LIN {X 0,Y 547.615,Z 386.436,A -85,B 0,C 180,E1 18147.997,E2 18147.997} C_VEL
LIN {X 0,Y 557.313,Z 399.518,A -85,B 0,C 180,E1 18145.988,E2 18145.988} C_VEL
LIN {X 0,Y 566.664,Z 412.794,A -85,B 0,C 180,E1 18144.201,E2 18144.201} C_VEL
LIN {X 0,Y 578.034,Z 429.679,A -85,B 0,C 180,E1 18142.193,E2 18142.193} C_VEL
LIN {X 0,Y 584.71,Z 440.377,A -85,B 0,C 180,E1 18141.078,E2 18141.078} C_VEL
LIN {X 0,Y 587.079,Z 454.76,A -85,B 0,C 180,E1 18140.491,E2 18140.491} C_VEL
LIN {X 0,Y 578.942,Z 687.19,A -85,B 0,C 180,E1 18137.176,E2 18137.176} C_VEL
LIN {X 0,Y 574.123,Z 831.147,A -85,B 0,C 180,E1 18135.139,E2 18135.139} C_VEL
LIN {X 0,Y 572.503,Z 855.718,A -85,B 0,C 180,E1 18134.679,E2 18134.679} C_VEL
LIN {X 0,Y 571.103,Z 863.307,A -85,B 0,C 180,E1 18134.585,E2 18134.585} C_VEL
LIN {X 0,Y 565.25,Z 881.378,A -85,B 0,C 180,E1 18134.516,E2 18134.516} C_VEL
LIN {X 0,Y 563.615,Z 888.829,A -85,B 0,C 180,E1 18134.375,E2 18134.375} C_VEL
LIN {X 0,Y 563.486,Z 889.888,A -85,B 0,C 180,E1 18134.344,E2 18134.344} C_VEL
LIN {X 0,Y 560.294,Z 914.057,A -85,B 0,C 180,E1 18133.468,E2 18133.468} C_VEL
LIN {X 0,Y 557.17,Z 934.515,A -85,B 0,C 180,E1 18132.575,E2 18132.575} C_VEL
LIN {X 0,Y 553.827,Z 954.3,A -85,B 0,C 180,E1 18131.566,E2 18131.566} C_VEL
LIN {X 0,Y 549.439,Z 977.967,A -85,B 0,C 180,E1 18130.152,E2 18130.152} C_VEL
LIN {X 0,Y 545.24,Z 998.451,A -85,B 0,C 180,E1 18128.707,E2 18128.707} C_VEL
LIN {X 0,Y 541.433,Z 1016.198,A -85,B 0,C 180,E1 18127.281,E2 18127.281} C_VEL
LIN {X 0,Y 536.891,Z 1036.776,A -85,B 0,C 180,E1 18125.394,E2 18125.394} C_VEL
LIN {X 0,Y 532.749,Z 1054.642,A -85,B 0,C 180,E1 18123.49,E2 18123.49} C_VEL
LIN {X 0,Y 529.257,Z 1069.696,A -85,B 0,C 180,E1 18121.682,E2 18121.682} C_VEL
LIN {X 0,Y 525.468,Z 1086.495,A -85,B 0,C 180,E1 18119.402,E2 18119.402} C_VEL
LIN {X 0,Y 522.072,Z 1101.673,A -85,B 0,C 180,E1 18116.995,E2 18116.995} C_VEL
LIN {X 0,Y 519.505,Z 1113.829,A -85,B 0,C 180,E1 18114.808,E2 18114.808} C_VEL
LIN {X 0,Y 517.039,Z 1126.95,A -85,B 0,C 180,E1 18112.13,E2 18112.13} C_VEL
LIN {X 0,Y 515.099,Z 1138.408,A -85,B 0,C 180,E1 18109.368,E2 18109.368} C_VEL
LIN {X 0,Y 513.904,Z 1147.043,A -85,B 0,C 180,E1 18106.969,E2 18106.969} C_VEL
LIN {X 0,Y 512.891,Z 1156.089,A -85,B 0,C 180,E1 18103.989,E2 18103.989} C_VEL
LIN {X 0,Y 512.347,Z 1162.485,A -85,B 0,C 180,E1 18101.368,E2 18101.368} C_VEL
LIN {X 0,Y 512.097,Z 1167.168,A -85,B 0,C 180,E1 18098.987,E2 18098.987} C_VEL
LIN {X 0,Y 511.954,Z 1171.379,A -85,B 0,C 180,E1 18096.167,E2 18096.167} C_VEL
LIN {X 0,Y 511.906,Z 1173.875,A -85,B 0,C 180,E1 18093.36,E2 18093.36} C_VEL
LIN {X 0,Y 511.909,Z 1174.869,A -85,B 0,C 180,E1 18091.007,E2 18091.007} C_VEL
LIN {X 0,Y 511.912,Z 1174.823,A -85,B 0,C 180,E1 18088.657,E2 18088.657} C_VEL
LIN {X 0,Y 511.915,Z 1173.467,A -85,B 0,C 180,E1 18085.856,E2 18085.856} C_VEL
LIN {X 0,Y 511.966,Z 1170.412,A -85,B 0,C 180,E1 18083.045,E2 18083.045} C_VEL
LIN {X 0,Y 512.119,Z 1166.721,A -85,B 0,C 180,E1 18080.674,E2 18080.674} C_VEL
LIN {X 0,Y 512.415,Z 1161.69,A -85,B 0,C 180,E1 18078.177,E2 18078.177} C_VEL
LIN {X 0,Y 513.117,Z 1153.749,A -85,B 0,C 180,E1 18075.095,E2 18075.095} C_VEL
LIN {X 0,Y 514.003,Z 1146.165,A -85,B 0,C 180,E1 18072.685,E2 18072.685} C_VEL
LIN {X 0,Y 515.264,Z 1137.342,A -85,B 0,C 180,E1 18070.267,E2 18070.267} C_VEL
LIN {X 0,Y 517.45,Z 1124.512,A -85,B 0,C 180,E1 18067.266,E2 18067.266} C_VEL
LIN {X 0,Y 519.656,Z 1113.054,A -85,B 0,C 180,E1 18064.957,E2 18064.957} C_VEL
LIN {X 0,Y 522.419,Z 1100.156,A -85,B 0,C 180,E1 18062.655,E2 18062.655} C_VEL
LIN {X 0,Y 526.146,Z 1083.341,A -85,B 0,C 180,E1 18060.065,E2 18060.065} C_VEL
LIN {X 0,Y 529.53,Z 1068.546,A -85,B 0,C 180,E1 18058.082,E2 18058.082} C_VEL
LIN {X 0,Y 533.173,Z 1052.881,A -85,B 0,C 180,E1 18056.218,E2 18056.218} C_VEL
LIN {X 0,Y 537.976,Z 1031.771,A -85,B 0,C 180,E1 18054.034,E2 18054.034} C_VEL
LIN {X 0,Y 541.945,Z 1013.857,A -85,B 0,C 180,E1 18052.428,E2 18052.428} C_VEL
LIN {X 0,Y 546.122,Z 994.411,A -85,B 0,C 180,E1 18050.895,E2 18050.895} C_VEL
LIN {X 0,Y 550.757,Z 971.131,A -85,B 0,C 180,E1 18049.327,E2 18049.327} C_VEL
LIN {X 0,Y 554.306,Z 951.689,A -85,B 0,C 180,E1 18048.202,E2 18048.202} C_VEL
LIN {X 0,Y 557.851,Z 930.54,A -85,B 0,C 180,E1 18047.146,E2 18047.146} C_VEL
LIN {X 0,Y 561.578,Z 905.044,A -85,B 0,C 180,E1 18046.093,E2 18046.093} C_VEL
LIN {X 0,Y 564.218,Z 883.465,A -85,B 0,C 180,E1 18045.369,E2 18045.369} C_VEL
LIN {X 0,Y 566.449,Z 861.689,A -85,B 0,C 180,E1 18044.778,E2 18044.778} C_VEL
LIN {X 0,Y 568.589,Z 834.181,A -85,B 0,C 180,E1 18044.222,E2 18044.222} C_VEL
LIN {X 0,Y 570.674,Z 778.593,A -85,B 0,C 180,E1 18043.415,E2 18043.415} C_VEL
LIN {X 0,Y 578.51,Z 553.659,A -85,B 0,C 180,E1 18040.214,E2 18040.214} C_VEL
LIN {X 0,Y 582.134,Z 455.512,A -85,B 0,C 180,E1 18038.781,E2 18038.781} C_VEL
LIN {X 0,Y 580.157,Z 444.764,A -85,B 0,C 180,E1 18038.302,E2 18038.302} C_VEL
LIN {X 0,Y 568.568,Z 426.659,A -85,B 0,C 180,E1 18036.283,E2 18036.283} C_VEL
LIN {X 0,Y 557.682,Z 410.932,A -85,B 0,C 180,E1 18034.232,E2 18034.232} C_VEL
LIN {X 0,Y 548.268,Z 397.906,A -85,B 0,C 180,E1 18032.3,E2 18032.3} C_VEL
LIN {X 0,Y 538.549,Z 384.76,A -85,B 0,C 180,E1 18030.086,E2 18030.086} C_VEL
LIN {X 0,Y 533.593,Z 375.407,A -85,B 0,C 180,E1 18027.814,E2 18027.814} C_VEL
LIN {X 0,Y 530.924,Z 370.532,A -85,B 0,C 180,E1 18026.509,E2 18026.509} C_VEL
LIN {X 0,Y 528.411,Z 365.874,A -85,B 0,C 180,E1 18025.199,E2 18025.199} C_VEL
LIN {X 0,Y 525.594,Z 360.858,A -85,B 0,C 180,E1 18023.666,E2 18023.666} C_VEL
LIN {X 0,Y 522.985,Z 356.145,A -85,B 0,C 180,E1 18022.126,E2 18022.126} C_VEL
LIN {X 0,Y 520.688,Z 352.401,A -85,B 0,C 180,E1 18020.743,E2 18020.743} C_VEL
LIN {X 0,Y 519.792,Z 350.773,A -85,B 0,C 180,E1 18020.141,E2 18020.141} C_VEL
LIN {X 0,Y 517.475,Z 347.05,A -85,B 0,C 180,E1 18018.592,E2 18018.592} C_VEL
LIN {X 0,Y 516.625,Z 345.409,A -85,B 0,C 180,E1 18017.923,E2 18017.923} C_VEL
LIN {X 0,Y 514.179,Z 341.868,A -85,B 0,C 180,E1 18016.131,E2 18016.131} C_VEL
LIN {X 0,Y 513.828,Z 340.405,A -85,B 0,C 180,E1 18015.462,E2 18015.462} C_VEL
LIN {X 0,Y 513.783,Z 340.151,A -85,B 0,C 180,E1 18012.133,E2 18012.133} C_VEL
LIN {X 0,Y 513.799,Z 340.19,A -85,B 0,C 180,E1 18008.618,E2 18008.618} C_VEL
LIN {X 0,Y 513.784,Z 340.162,A -85,B 0,C 180,E1 18005.136,E2 18005.136} C_VEL
LIN {X 0,Y 513.798,Z 340.17,A -85,B 0,C 180,E1 18001.784,E2 18001.784} C_VEL
LIN {X 0,Y 513.802,Z 340.182,A -85,B 0,C 180,E1 17998.216,E2 17998.216} C_VEL
LIN {X 0,Y 513.777,Z 340.156,A -85,B 0,C 180,E1 17994.752,E2 17994.752} C_VEL
LIN {X 0,Y 513.782,Z 340.219,A -85,B 0,C 180,E1 17991.156,E2 17991.156} C_VEL
LIN {X 0,Y 513.798,Z 340.148,A -85,B 0,C 180,E1 17987.639,E2 17987.639} C_VEL
LIN {X 0,Y 513.881,Z 340.659,A -85,B 0,C 180,E1 17985.959,E2 17985.959} C_VEL
LIN {X 0,Y 515.526,Z 344.286,A -85,B 0,C 180,E1 17984.36,E2 17984.36} C_VEL
LIN {X 0,Y 517.264,Z 346.356,A -85,B 0,C 180,E1 17983.26,E2 17983.26} C_VEL
LIN {X 0,Y 519.227,Z 350.069,A -85,B 0,C 180,E1 17981.822,E2 17981.822} C_VEL
LIN {X 0,Y 520.553,Z 351.834,A -85,B 0,C 180,E1 17981.057,E2 17981.057} C_VEL
LIN {X 0,Y 522.599,Z 355.65,A -85,B 0,C 180,E1 17979.738,E2 17979.738} C_VEL
LIN {X 0,Y 523.786,Z 357.449,A -85,B 0,C 180,E1 17979.085,E2 17979.085} C_VEL
LIN {X 0,Y 526.164,Z 361.41,A -85,B 0,C 180,E1 17977.78,E2 17977.78} C_VEL
LIN {X 0,Y 527.603,Z 363.761,A -85,B 0,C 180,E1 17977.227,E2 17977.227} C_VEL
LIN {X 0,Y 532.292,Z 368.989,A -85,B 0,C 180,E1 17976.003,E2 17976.003} C_VEL
LIN {X 0,Y 536.471,Z 373.737,A -85,B 0,C 180,E1 17974.97,E2 17974.97} C_VEL
LIN {X 0,Y 547.139,Z 386.885,A -85,B 0,C 180,E1 17972.52,E2 17972.52} C_VEL
LIN {X 0,Y 558.265,Z 401.008,A -85,B 0,C 180,E1 17970.226,E2 17970.226} C_VEL
LIN {X 0,Y 569.426,Z 416.229,A -85,B 0,C 180,E1 17968.122,E2 17968.122} C_VEL
LIN {X 0,Y 580.784,Z 432.397,A -85,B 0,C 180,E1 17966.155,E2 17966.155} C_VEL
LIN {X 0,Y 586.451,Z 441.212,A -85,B 0,C 180,E1 17965.219,E2 17965.219} C_VEL
LIN {X 0,Y 577.985,Z 650.891,A -85,B 0,C 180,E1 17962.065,E2 17962.065} C_VEL
LIN {X 0,Y 571.099,Z 826.33,A -85,B 0,C 180,E1 17959.44,E2 17959.44} C_VEL
LIN {X 0,Y 569.144,Z 853.345,A -85,B 0,C 180,E1 17958.924,E2 17958.924} C_VEL
LIN {X 0,Y 566.435,Z 879.926,A -85,B 0,C 180,E1 17958.223,E2 17958.223} C_VEL
LIN {X 0,Y 563.88,Z 901.17,A -85,B 0,C 180,E1 17957.532,E2 17957.532} C_VEL
LIN {X 0,Y 561.044,Z 922.127,A -85,B 0,C 180,E1 17956.72,E2 17956.72} C_VEL
LIN {X 0,Y 557.782,Z 943.866,A -85,B 0,C 180,E1 17955.736,E2 17955.736} C_VEL
LIN {X 0,Y 553.31,Z 970.62,A -85,B 0,C 180,E1 17954.306,E2 17954.306} C_VEL
LIN {X 0,Y 549.568,Z 991.286,A -85,B 0,C 180,E1 17953.021,E2 17953.021} C_VEL
LIN {X 0,Y 545.927,Z 1010.645,A -85,B 0,C 180,E1 17951.67,E2 17951.67} C_VEL
LIN {X 0,Y 541.854,Z 1031.6,A -85,B 0,C 180,E1 17950.021,E2 17950.021} C_VEL
LIN {X 0,Y 537.242,Z 1054.179,A -85,B 0,C 180,E1 17947.974,E2 17947.974} C_VEL
LIN {X 0,Y 533.599,Z 1071.666,A -85,B 0,C 180,E1 17946.175,E2 17946.175} C_VEL
LIN {X 0,Y 530.321,Z 1087.231,A -85,B 0,C 180,E1 17944.38,E2 17944.38} C_VEL
LIN {X 0,Y 527.005,Z 1103.09,A -85,B 0,C 180,E1 17942.346,E2 17942.346} C_VEL
LIN {X 0,Y 523.228,Z 1121.849,A -85,B 0,C 180,E1 17939.598,E2 17939.598} C_VEL
LIN {X 0,Y 520.656,Z 1134.443,A -85,B 0,C 180,E1 17937.445,E2 17937.445} C_VEL
LIN {X 0,Y 518.457,Z 1145.98,A -85,B 0,C 180,E1 17935.227,E2 17935.227} C_VEL
LIN {X 0,Y 516.576,Z 1156.883,A -85,B 0,C 180,E1 17932.875,E2 17932.875} C_VEL
LIN {X 0,Y 514.817,Z 1168.634,A -85,B 0,C 180,E1 17929.988,E2 17929.988} C_VEL
LIN {X 0,Y 513.537,Z 1178.567,A -85,B 0,C 180,E1 17927.057,E2 17927.057} C_VEL
LIN {X 0,Y 512.82,Z 1185.755,A -85,B 0,C 180,E1 17924.567,E2 17924.567} C_VEL
LIN {X 0,Y 512.357,Z 1191.694,A -85,B 0,C 180,E1 17922.114,E2 17922.114} C_VEL
LIN {X 0,Y 512.077,Z 1197.139,A -85,B 0,C 180,E1 17919.327,E2 17919.327} C_VEL
LIN {X 0,Y 511.947,Z 1201.479,A -85,B 0,C 180,E1 17916.206,E2 17916.206} C_VEL
LIN {X 0,Y 511.913,Z 1203.76,A -85,B 0,C 180,E1 17913.583,E2 17913.583} C_VEL
LIN {X 0,Y 511.914,Z 1204.758,A -85,B 0,C 180,E1 17911.231,E2 17911.231} C_VEL
LIN {X 0,Y 511.909,Z 1204.803,A -85,B 0,C 180,E1 17908.993,E2 17908.993} C_VEL
LIN {X 0,Y 511.916,Z 1203.895,A -85,B 0,C 180,E1 17906.641,E2 17906.641} C_VEL
LIN {X 0,Y 511.939,Z 1201.857,A -85,B 0,C 180,E1 17904.171,E2 17904.171} C_VEL
LIN {X 0,Y 512.032,Z 1198.398,A -85,B 0,C 180,E1 17901.465,E2 17901.465} C_VEL
LIN {X 0,Y 512.307,Z 1192.592,A -85,B 0,C 180,E1 17898.289,E2 17898.289} C_VEL
LIN {X 0,Y 512.769,Z 1186.358,A -85,B 0,C 180,E1 17895.662,E2 17895.662} C_VEL
LIN {X 0,Y 513.436,Z 1179.5,A -85,B 0,C 180,E1 17893.248,E2 17893.248} C_VEL
LIN {X 0,Y 514.41,Z 1171.481,A -85,B 0,C 180,E1 17890.823,E2 17890.823} C_VEL
LIN {X 0,Y 516.054,Z 1160.38,A -85,B 0,C 180,E1 17887.921,E2 17887.921} C_VEL
LIN {X 0,Y 518.198,Z 1147.491,A -85,B 0,C 180,E1 17885.08,E2 17885.08} C_VEL
LIN {X 0,Y 520.397,Z 1135.714,A -85,B 0,C 180,E1 17882.788,E2 17882.788} C_VEL
LIN {X 0,Y 522.855,Z 1123.631,A -85,B 0,C 180,E1 17880.688,E2 17880.688} C_VEL
LIN {X 0,Y 525.936,Z 1108.474,A -85,B 0,C 180,E1 17878.4,E2 17878.4} C_VEL
LIN {X 0,Y 529.914,Z 1089.158,A -85,B 0,C 180,E1 17875.851,E2 17875.851} C_VEL
LIN {X 0,Y 533.373,Z 1072.717,A -85,B 0,C 180,E1 17873.94,E2 17873.94} C_VEL
LIN {X 0,Y 536.841,Z 1056.057,A -85,B 0,C 180,E1 17872.21,E2 17872.21} C_VEL
LIN {X 0,Y 540.923,Z 1036.267,A -85,B 0,C 180,E1 17870.378,E2 17870.378} C_VEL
LIN {X 0,Y 545.441,Z 1013.284,A -85,B 0,C 180,E1 17868.525,E2 17868.525} C_VEL
LIN {X 0,Y 549.262,Z 992.967,A -85,B 0,C 180,E1 17867.091,E2 17867.091} C_VEL
LIN {X 0,Y 552.658,Z 974.273,A -85,B 0,C 180,E1 17865.912,E2 17865.912} C_VEL
LIN {X 0,Y 556.045,Z 954.475,A -85,B 0,C 180,E1 17864.802,E2 17864.802} C_VEL
LIN {X 0,Y 560.133,Z 928.662,A -85,B 0,C 180,E1 17863.553,E2 17863.553} C_VEL
LIN {X 0,Y 563.499,Z 904.146,A -85,B 0,C 180,E1 17862.576,E2 17862.576} C_VEL
LIN {X 0,Y 566.099,Z 882.845,A -85,B 0,C 180,E1 17861.866,E2 17861.866} C_VEL
LIN {X 0,Y 568.32,Z 861.452,A -85,B 0,C 180,E1 17861.276,E2 17861.276} C_VEL
LIN {X 0,Y 570.444,Z 836.682,A -85,B 0,C 180,E1 17860.738,E2 17860.738} C_VEL
LIN {X 0,Y 572.278,Z 799.543,A -85,B 0,C 180,E1 17860.147,E2 17860.147} C_VEL
LIN {X 0,Y 581.073,Z 573.004,A -85,B 0,C 180,E1 17856.77,E2 17856.77} C_VEL
LIN {X 0,Y 586.338,Z 440.884,A -85,B 0,C 180,E1 17854.765,E2 17854.765} C_VEL
LIN {X 0,Y 573.946,Z 422.524,A -85,B 0,C 180,E1 17852.688,E2 17852.688} C_VEL
LIN {X 0,Y 560.652,Z 404.185,A -85,B 0,C 180,E1 17850.253,E2 17850.253} C_VEL
LIN {X 0,Y 549.148,Z 389.385,A -85,B 0,C 180,E1 17847.931,E2 17847.931} C_VEL
LIN {X 0,Y 540.25,Z 378.476,A -85,B 0,C 180,E1 17845.958,E2 17845.958} C_VEL
LIN {X 0,Y 535.753,Z 373.1,A -85,B 0,C 180,E1 17844.889,E2 17844.889} C_VEL
LIN {X 0,Y 530.64,Z 367.097,A -85,B 0,C 180,E1 17843.604,E2 17843.604} C_VEL
LIN {X 0,Y 526.894,Z 362.698,A -85,B 0,C 180,E1 17842.6,E2 17842.6} C_VEL
LIN {X 0,Y 525.611,Z 360.76,A -85,B 0,C 180,E1 17842.01,E2 17842.01} C_VEL
LIN {X 0,Y 522.947,Z 356.065,A -85,B 0,C 180,E1 17840.481,E2 17840.481} C_VEL
LIN {X 0,Y 520.615,Z 352.049,A -85,B 0,C 180,E1 17839.057,E2 17839.057} C_VEL
LIN {X 0,Y 519.326,Z 350.185,A -85,B 0,C 180,E1 17838.291,E2 17838.291} C_VEL
LIN {X 0,Y 517.303,Z 346.516,A -85,B 0,C 180,E1 17836.854,E2 17836.854} C_VEL
LIN {X 0,Y 514.208,Z 341.953,A -85,B 0,C 180,E1 17834.643,E2 17834.643} C_VEL
LIN {X 0,Y 513.827,Z 340.372,A -85,B 0,C 180,E1 17833.906,E2 17833.906} C_VEL
LIN {X 0,Y 513.79,Z 340.174,A -85,B 0,C 180,E1 17830.541,E2 17830.541} C_VEL
LIN {X 0,Y 513.768,Z 340.161,A -85,B 0,C 180,E1 17827.155,E2 17827.155} C_VEL
LIN {X 0,Y 513.801,Z 340.202,A -85,B 0,C 180,E1 17823.682,E2 17823.682} C_VEL
LIN {X 0,Y 513.801,Z 340.146,A -85,B 0,C 180,E1 17820.223,E2 17820.223} C_VEL
LIN {X 0,Y 513.792,Z 340.231,A -85,B 0,C 180,E1 17816.653,E2 17816.653} C_VEL
LIN {X 0,Y 513.791,Z 340.145,A -85,B 0,C 180,E1 17813.07,E2 17813.07} C_VEL
LIN {X 0,Y 513.793,Z 340.196,A -85,B 0,C 180,E1 17809.686,E2 17809.686} C_VEL
LIN {X 0,Y 513.802,Z 340.161,A -85,B 0,C 180,E1 17806.151,E2 17806.151} C_VEL
LIN {X 0,Y 513.87,Z 340.641,A -85,B 0,C 180,E1 17804.192,E2 17804.192} C_VEL
LIN {X 0,Y 515.654,Z 344.375,A -85,B 0,C 180,E1 17802.509,E2 17802.509} C_VEL
LIN {X 0,Y 517.322,Z 346.603,A -85,B 0,C 180,E1 17801.403,E2 17801.403} C_VEL
LIN {X 0,Y 519.533,Z 350.49,A -85,B 0,C 180,E1 17799.848,E2 17799.848} C_VEL
LIN {X 0,Y 520.597,Z 352.15,A -85,B 0,C 180,E1 17799.187,E2 17799.187} C_VEL
LIN {X 0,Y 522.717,Z 355.851,A -85,B 0,C 180,E1 17797.862,E2 17797.862} C_VEL
LIN {X 0,Y 523.674,Z 357.409,A -85,B 0,C 180,E1 17797.313,E2 17797.313} C_VEL
LIN {X 0,Y 526.033,Z 361.382,A -85,B 0,C 180,E1 17795.998,E2 17795.998} C_VEL
LIN {X 0,Y 528.882,Z 366.467,A -85,B 0,C 180,E1 17794.466,E2 17794.466} C_VEL
LIN {X 0,Y 532.283,Z 373.059,A -85,B 0,C 180,E1 17792.688,E2 17792.688} C_VEL
LIN {X 0,Y 535.175,Z 378.463,A -85,B 0,C 180,E1 17791.304,E2 17791.304} C_VEL
LIN {X 0,Y 539.213,Z 385.657,A -85,B 0,C 180,E1 17789.617,E2 17789.617} C_VEL
LIN {X 0,Y 551.212,Z 401.903,A -85,B 0,C 180,E1 17786.968,E2 17786.968} C_VEL
LIN {X 0,Y 562.347,Z 417.59,A -85,B 0,C 180,E1 17784.761,E2 17784.761} C_VEL
LIN {X 0,Y 574.295,Z 435.493,A -85,B 0,C 180,E1 17782.597,E2 17782.597} C_VEL
LIN {X 0,Y 580.363,Z 445.427,A -85,B 0,C 180,E1 17781.556,E2 17781.556} C_VEL
LIN {X 0,Y 582.161,Z 456.877,A -85,B 0,C 180,E1 17781.089,E2 17781.089} C_VEL
LIN {X 0,Y 573.691,Z 688.655,A -85,B 0,C 180,E1 17777.763,E2 17777.763} C_VEL
LIN {X 0,Y 568.71,Z 831.17,A -85,B 0,C 180,E1 17775.733,E2 17775.733} C_VEL
LIN {X 0,Y 566.835,Z 857.684,A -85,B 0,C 180,E1 17775.226,E2 17775.226} C_VEL
LIN {X 0,Y 564.428,Z 881.502,A -85,B 0,C 180,E1 17774.596,E2 17774.596} C_VEL
LIN {X 0,Y 563.486,Z 889.888,A -85,B 0,C 180,E1 17774.344,E2 17774.344} C_VEL
LIN {X 0,Y 561.926,Z 897.311,A -85,B 0,C 180,E1 17774.175,E2 17774.175} C_VEL
LIN {X 0,Y 555.07,Z 916.056,A -85,B 0,C 180,E1 17773.908,E2 17773.908} C_VEL
LIN {X 0,Y 553.301,Z 923.248,A -85,B 0,C 180,E1 17773.683,E2 17773.683} C_VEL
LIN {X 0,Y 549.082,Z 948.317,A -85,B 0,C 180,E1 17772.48,E2 17772.48} C_VEL
LIN {X 0,Y 545.579,Z 966.984,A -85,B 0,C 180,E1 17771.422,E2 17771.422} C_VEL
LIN {X 0,Y 541.856,Z 985.41,A -85,B 0,C 180,E1 17770.23,E2 17770.23} C_VEL
LIN {X 0,Y 537.275,Z 1006.886,A -85,B 0,C 180,E1 17768.636,E2 17768.636} C_VEL
LIN {X 0,Y 532.651,Z 1026.853,A -85,B 0,C 180,E1 17766.9,E2 17766.9} C_VEL
LIN {X 0,Y 528.789,Z 1043.181,A -85,B 0,C 180,E1 17765.288,E2 17765.288} C_VEL
LIN {X 0,Y 524.781,Z 1059.88,A -85,B 0,C 180,E1 17763.431,E2 17763.431} C_VEL
LIN {X 0,Y 520.222,Z 1078.787,A -85,B 0,C 180,E1 17761.004,E2 17761.004} C_VEL
LIN {X 0,Y 517.049,Z 1092.182,A -85,B 0,C 180,E1 17759.038,E2 17759.038} C_VEL
LIN {X 0,Y 514.142,Z 1104.884,A -85,B 0,C 180,E1 17756.945,E2 17756.945} C_VEL
LIN {X 0,Y 511.093,Z 1119.129,A -85,B 0,C 180,E1 17754.257,E2 17754.257} C_VEL
LIN {X 0,Y 508.715,Z 1131.091,A -85,B 0,C 180,E1 17751.612,E2 17751.612} C_VEL
LIN {X 0,Y 506.97,Z 1141.408,A -85,B 0,C 180,E1 17748.991,E2 17748.991} C_VEL
LIN {X 0,Y 505.556,Z 1151.446,A -85,B 0,C 180,E1 17745.957,E2 17745.957} C_VEL
LIN {X 0,Y 504.798,Z 1158.345,A -85,B 0,C 180,E1 17743.452,E2 17743.452} C_VEL
LIN {X 0,Y 504.312,Z 1164.264,A -85,B 0,C 180,E1 17740.857,E2 17740.857} C_VEL
LIN {X 0,Y 504.026,Z 1169.625,A -85,B 0,C 180,E1 17737.753,E2 17737.753} C_VEL
LIN {X 0,Y 503.934,Z 1172.536,A -85,B 0,C 180,E1 17735.351,E2 17735.351} C_VEL
LIN {X 0,Y 503.911,Z 1174.393,A -85,B 0,C 180,E1 17732.957,E2 17732.957} C_VEL
LIN {X 0,Y 503.899,Z 1175.23,A -85,B 0,C 180,E1 17730.455,E2 17730.455} C_VEL
LIN {X 0,Y 503.917,Z 1174.712,A -85,B 0,C 180,E1 17727.498,E2 17727.498} C_VEL
LIN {X 0,Y 503.93,Z 1172.881,A -85,B 0,C 180,E1 17724.916,E2 17724.916} C_VEL
LIN {X 0,Y 504.007,Z 1170.212,A -85,B 0,C 180,E1 17722.591,E2 17722.591} C_VEL
LIN {X 0,Y 504.172,Z 1166.4,A -85,B 0,C 180,E1 17720.18,E2 17720.18} C_VEL
LIN {X 0,Y 504.65,Z 1160.014,A -85,B 0,C 180,E1 17717.118,E2 17717.118} C_VEL
LIN {X 0,Y 505.371,Z 1152.99,A -85,B 0,C 180,E1 17714.482,E2 17714.482} C_VEL
LIN {X 0,Y 506.351,Z 1145.373,A -85,B 0,C 180,E1 17712.059,E2 17712.059} C_VEL
LIN {X 0,Y 508.06,Z 1134.887,A -85,B 0,C 180,E1 17709.201,E2 17709.201} C_VEL
LIN {X 0,Y 510.221,Z 1123.167,A -85,B 0,C 180,E1 17706.513,E2 17706.513} C_VEL
LIN {X 0,Y 512.497,Z 1112.378,A -85,B 0,C 180,E1 17704.335,E2 17704.335} C_VEL
LIN {X 0,Y 515.763,Z 1097.93,A -85,B 0,C 180,E1 17701.769,E2 17701.769} C_VEL
LIN {X 0,Y 519.496,Z 1081.83,A -85,B 0,C 180,E1 17699.333,E2 17699.333} C_VEL
LIN {X 0,Y 523.016,Z 1067.197,A -85,B 0,C 180,E1 17697.377,E2 17697.377} C_VEL
LIN {X 0,Y 527.477,Z 1048.815,A -85,B 0,C 180,E1 17695.21,E2 17695.21} C_VEL
LIN {X 0,Y 531.938,Z 1029.877,A -85,B 0,C 180,E1 17693.292,E2 17693.292} C_VEL
LIN {X 0,Y 535.973,Z 1012.393,A -85,B 0,C 180,E1 17691.731,E2 17691.731} C_VEL
LIN {X 0,Y 540.847,Z 990.479,A -85,B 0,C 180,E1 17690.027,E2 17690.027} C_VEL
LIN {X 0,Y 545.016,Z 969.95,A -85,B 0,C 180,E1 17688.666,E2 17688.666} C_VEL
LIN {X 0,Y 548.569,Z 951.139,A -85,B 0,C 180,E1 17687.579,E2 17687.579} C_VEL
LIN {X 0,Y 552.227,Z 930.028,A -85,B 0,C 180,E1 17686.525,E2 17686.525} C_VEL
LIN {X 0,Y 556.069,Z 904.457,A -85,B 0,C 180,E1 17685.472,E2 17685.472} C_VEL
LIN {X 0,Y 558.732,Z 883.406,A -85,B 0,C 180,E1 17684.765,E2 17684.765} C_VEL
LIN {X 0,Y 561.021,Z 861.745,A -85,B 0,C 180,E1 17684.175,E2 17684.175} C_VEL
LIN {X 0,Y 563.232,Z 834.254,A -85,B 0,C 180,E1 17683.617,E2 17683.617} C_VEL
LIN {X 0,Y 565.381,Z 779.266,A -85,B 0,C 180,E1 17682.814,E2 17682.814} C_VEL
LIN {X 0,Y 573.565,Z 554.307,A -85,B 0,C 180,E1 17679.592,E2 17679.592} C_VEL
LIN {X 0,Y 577.289,Z 457.505,A -85,B 0,C 180,E1 17678.169,E2 17678.169} C_VEL
LIN {X 0,Y 575.87,Z 449.769,A -85,B 0,C 180,E1 17677.817,E2 17677.817} C_VEL
LIN {X 0,Y 564.927,Z 432.548,A -85,B 0,C 180,E1 17675.863,E2 17675.863} C_VEL
LIN {X 0,Y 553.282,Z 415.457,A -85,B 0,C 180,E1 17673.605,E2 17673.605} C_VEL
LIN {X 0,Y 542.975,Z 401.194,A -85,B 0,C 180,E1 17671.409,E2 17671.409} C_VEL
LIN {X 0,Y 535.047,Z 390.731,A -85,B 0,C 180,E1 17669.562,E2 17669.562} C_VEL
LIN {X 0,Y 529.713,Z 383.472,A -85,B 0,C 180,E1 17668.158,E2 17668.158} C_VEL
LIN {X 0,Y 526.151,Z 376.878,A -85,B 0,C 180,E1 17666.404,E2 17666.404} C_VEL
LIN {X 0,Y 523.427,Z 371.904,A -85,B 0,C 180,E1 17664.972,E2 17664.972} C_VEL
LIN {X 0,Y 520.872,Z 367.215,A -85,B 0,C 180,E1 17663.534,E2 17663.534} C_VEL
LIN {X 0,Y 518.284,Z 362.525,A -85,B 0,C 180,E1 17661.979,E2 17661.979} C_VEL
LIN {X 0,Y 515.983,Z 358.591,A -85,B 0,C 180,E1 17660.533,E2 17660.533} C_VEL
LIN {X 0,Y 514.547,Z 356.484,A -85,B 0,C 180,E1 17659.644,E2 17659.644} C_VEL
LIN {X 0,Y 512.187,Z 352.036,A -85,B 0,C 180,E1 17657.848,E2 17657.848} C_VEL
LIN {X 0,Y 509.676,Z 348.267,A -85,B 0,C 180,E1 17655.942,E2 17655.942} C_VEL
LIN {X 0,Y 508.881,Z 346.589,A -85,B 0,C 180,E1 17655.149,E2 17655.149} C_VEL
LIN {X 0,Y 506.174,Z 342.599,A -85,B 0,C 180,E1 17652.624,E2 17652.624} C_VEL
LIN {X 0,Y 505.882,Z 341.339,A -85,B 0,C 180,E1 17651.747,E2 17651.747} C_VEL
LIN {X 0,Y 505.85,Z 341.161,A -85,B 0,C 180,E1 17648.182,E2 17648.182} C_VEL
LIN {X 0,Y 505.857,Z 341.161,A -85,B 0,C 180,E1 17644.648,E2 17644.648} C_VEL
LIN {X 0,Y 505.842,Z 341.142,A -85,B 0,C 180,E1 17641.133,E2 17641.133} C_VEL
LIN {X 0,Y 505.861,Z 341.193,A -85,B 0,C 180,E1 17637.621,E2 17637.621} C_VEL
LIN {X 0,Y 505.859,Z 341.133,A -85,B 0,C 180,E1 17634.1,E2 17634.1} C_VEL
LIN {X 0,Y 505.843,Z 341.22,A -85,B 0,C 180,E1 17630.672,E2 17630.672} C_VEL
LIN {X 0,Y 505.944,Z 341.729,A -85,B 0,C 180,E1 17629.467,E2 17629.467} C_VEL
LIN {X 0,Y 508.107,Z 345.813,A -85,B 0,C 180,E1 17627.036,E2 17627.036} C_VEL
LIN {X 0,Y 509.523,Z 347.642,A -85,B 0,C 180,E1 17625.916,E2 17625.916} C_VEL
LIN {X 0,Y 511.304,Z 351.116,A -85,B 0,C 180,E1 17624.343,E2 17624.343} C_VEL
LIN {X 0,Y 512.826,Z 353.045,A -85,B 0,C 180,E1 17623.344,E2 17623.344} C_VEL
LIN {X 0,Y 514.804,Z 356.703,A -85,B 0,C 180,E1 17621.895,E2 17621.895} C_VEL
LIN {X 0,Y 516.071,Z 358.556,A -85,B 0,C 180,E1 17621.121,E2 17621.121} C_VEL
LIN {X 0,Y 518.37,Z 362.541,A -85,B 0,C 180,E1 17619.683,E2 17619.683} C_VEL
LIN {X 0,Y 519.469,Z 364.091,A -85,B 0,C 180,E1 17619.228,E2 17619.228} C_VEL
LIN {X 0,Y 523.232,Z 368.386,A -85,B 0,C 180,E1 17618.121,E2 17618.121} C_VEL
LIN {X 0,Y 525.046,Z 370.504,A -85,B 0,C 180,E1 17617.612,E2 17617.612} C_VEL
LIN {X 0,Y 528.998,Z 374.884,A -85,B 0,C 180,E1 17616.554,E2 17616.554} C_VEL
LIN {X 0,Y 533.86,Z 380.72,A -85,B 0,C 180,E1 17615.313,E2 17615.313} C_VEL
LIN {X 0,Y 543.767,Z 392.902,A -85,B 0,C 180,E1 17612.987,E2 17612.987} C_VEL
LIN {X 0,Y 555.294,Z 407.713,A -85,B 0,C 180,E1 17610.556,E2 17610.556} C_VEL
LIN {X 0,Y 566.339,Z 422.946,A -85,B 0,C 180,E1 17608.434,E2 17608.434} C_VEL
LIN {X 0,Y 577.336,Z 438.765,A -85,B 0,C 180,E1 17606.492,E2 17606.492} C_VEL
LIN {X 0,Y 581.476,Z 445.523,A -85,B 0,C 180,E1 17605.787,E2 17605.787} C_VEL
LIN {X 0,Y 572.659,Z 655.383,A -85,B 0,C 180,E1 17602.612,E2 17602.612} C_VEL
LIN {X 0,Y 565.669,Z 826.381,A -85,B 0,C 180,E1 17600.036,E2 17600.036} C_VEL
LIN {X 0,Y 563.64,Z 853.433,A -85,B 0,C 180,E1 17599.516,E2 17599.516} C_VEL
LIN {X 0,Y 560.83,Z 880.022,A -85,B 0,C 180,E1 17598.811,E2 17598.811} C_VEL
LIN {X 0,Y 558.134,Z 901.614,A -85,B 0,C 180,E1 17598.103,E2 17598.103} C_VEL
LIN {X 0,Y 555.199,Z 922.47,A -85,B 0,C 180,E1 17597.288,E2 17597.288} C_VEL
LIN {X 0,Y 551.634,Z 945.265,A -85,B 0,C 180,E1 17596.245,E2 17596.245} C_VEL
LIN {X 0,Y 547.062,Z 971.236,A -85,B 0,C 180,E1 17594.833,E2 17594.833} C_VEL
LIN {X 0,Y 543.257,Z 991.241,A -85,B 0,C 180,E1 17593.572,E2 17593.572} C_VEL
LIN {X 0,Y 539.291,Z 1011.128,A -85,B 0,C 180,E1 17592.157,E2 17592.157} C_VEL
LIN {X 0,Y 534.467,Z 1034.85,A -85,B 0,C 180,E1 17590.244,E2 17590.244} C_VEL
LIN {X 0,Y 530.117,Z 1055.133,A -85,B 0,C 180,E1 17588.355,E2 17588.355} C_VEL
LIN {X 0,Y 526.586,Z 1071.464,A -85,B 0,C 180,E1 17586.653,E2 17586.653} C_VEL
LIN {X 0,Y 523.211,Z 1087.039,A -85,B 0,C 180,E1 17584.848,E2 17584.848} C_VEL
LIN {X 0,Y 519.842,Z 1102.482,A -85,B 0,C 180,E1 17582.847,E2 17582.847} C_VEL
LIN {X 0,Y 515.936,Z 1120.925,A -85,B 0,C 180,E1 17580.128,E2 17580.128} C_VEL
LIN {X 0,Y 513.073,Z 1134.938,A -85,B 0,C 180,E1 17577.759,E2 17577.759} C_VEL
LIN {X 0,Y 511.115,Z 1144.874,A -85,B 0,C 180,E1 17575.855,E2 17575.855} C_VEL
LIN {X 0,Y 509.09,Z 1155.764,A -85,B 0,C 180,E1 17573.497,E2 17573.497} C_VEL
LIN {X 0,Y 507.478,Z 1165.432,A -85,B 0,C 180,E1 17571.134,E2 17571.134} C_VEL
LIN {X 0,Y 506.058,Z 1175.532,A -85,B 0,C 180,E1 17568.31,E2 17568.31} C_VEL
LIN {X 0,Y 504.987,Z 1184.842,A -85,B 0,C 180,E1 17565.151,E2 17565.151} C_VEL
LIN {X 0,Y 504.432,Z 1191.064,A -85,B 0,C 180,E1 17562.594,E2 17562.594} C_VEL
LIN {X 0,Y 504.136,Z 1196.103,A -85,B 0,C 180,E1 17560.051,E2 17560.051} C_VEL
LIN {X 0,Y 503.987,Z 1200.154,A -85,B 0,C 180,E1 17557.409,E2 17557.409} C_VEL
LIN {X 0,Y 503.919,Z 1203.349,A -85,B 0,C 180,E1 17554.324,E2 17554.324} C_VEL
LIN {X 0,Y 503.908,Z 1204.69,A -85,B 0,C 180,E1 17551.592,E2 17551.592} C_VEL
LIN {X 0,Y 503.901,Z 1204.848,A -85,B 0,C 180,E1 17549.204,E2 17549.204} C_VEL
LIN {X 0,Y 503.917,Z 1204.029,A -85,B 0,C 180,E1 17546.815,E2 17546.815} C_VEL
LIN {X 0,Y 503.934,Z 1202.196,A -85,B 0,C 180,E1 17544.42,E2 17544.42} C_VEL
LIN {X 0,Y 504.009,Z 1199.353,A -85,B 0,C 180,E1 17542.017,E2 17542.017} C_VEL
LIN {X 0,Y 504.178,Z 1195.276,A -85,B 0,C 180,E1 17539.487,E2 17539.487} C_VEL
LIN {X 0,Y 504.596,Z 1189.282,A -85,B 0,C 180,E1 17536.594,E2 17536.594} C_VEL
LIN {X 0,Y 505.386,Z 1180.912,A -85,B 0,C 180,E1 17533.447,E2 17533.447} C_VEL
LIN {X 0,Y 506.366,Z 1173.099,A -85,B 0,C 180,E1 17530.985,E2 17530.985} C_VEL
LIN {X 0,Y 507.617,Z 1164.516,A -85,B 0,C 180,E1 17528.629,E2 17528.629} C_VEL
LIN {X 0,Y 509.278,Z 1154.739,A -85,B 0,C 180,E1 17526.266,E2 17526.266} C_VEL
LIN {X 0,Y 511.858,Z 1141.395,A -85,B 0,C 180,E1 17523.427,E2 17523.427} C_VEL
LIN {X 0,Y 514.715,Z 1126.732,A -85,B 0,C 180,E1 17520.818,E2 17520.818} C_VEL
LIN {X 0,Y 517.644,Z 1112.766,A -85,B 0,C 180,E1 17518.625,E2 17518.625} C_VEL
LIN {X 0,Y 520.649,Z 1098.802,A -85,B 0,C 180,E1 17516.658,E2 17516.658} C_VEL
LIN {X 0,Y 523.905,Z 1083.899,A -85,B 0,C 180,E1 17514.771,E2 17514.771} C_VEL
LIN {X 0,Y 528.266,Z 1063.863,A -85,B 0,C 180,E1 17512.517,E2 17512.517} C_VEL
LIN {X 0,Y 532.563,Z 1043.568,A -85,B 0,C 180,E1 17510.541,E2 17510.541} C_VEL
LIN {X 0,Y 536.303,Z 1025.615,A -85,B 0,C 180,E1 17508.984,E2 17508.984} C_VEL
LIN {X 0,Y 540.607,Z 1004.613,A -85,B 0,C 180,E1 17507.356,E2 17507.356} C_VEL
LIN {X 0,Y 545.624,Z 978.991,A -85,B 0,C 180,E1 17505.636,E2 17505.636} C_VEL
LIN {X 0,Y 549.247,Z 958.936,A -85,B 0,C 180,E1 17504.47,E2 17504.47} C_VEL
LIN {X 0,Y 552.738,Z 938.175,A -85,B 0,C 180,E1 17503.414,E2 17503.414} C_VEL
LIN {X 0,Y 556.16,Z 915.89,A -85,B 0,C 180,E1 17502.438,E2 17502.438} C_VEL
LIN {X 0,Y 559.964,Z 887.346,A -85,B 0,C 180,E1 17501.413,E2 17501.413} C_VEL
LIN {X 0,Y 562.495,Z 864.435,A -85,B 0,C 180,E1 17500.759,E2 17500.759} C_VEL
LIN {X 0,Y 564.468,Z 842.977,A -85,B 0,C 180,E1 17500.27,E2 17500.27} C_VEL
LIN {X 0,Y 566.048,Z 819.294,A -85,B 0,C 180,E1 17499.849,E2 17499.849} C_VEL
LIN {X 0,Y 575.004,Z 598.092,A -85,B 0,C 180,E1 17496.526,E2 17496.526} C_VEL
LIN {X 0,Y 581.352,Z 445.027,A -85,B 0,C 180,E1 17494.194,E2 17494.194} C_VEL
LIN {X 0,Y 569.219,Z 426.931,A -85,B 0,C 180,E1 17492.098,E2 17492.098} C_VEL
LIN {X 0,Y 556.953,Z 410.009,A -85,B 0,C 180,E1 17489.792,E2 17489.792} C_VEL
LIN {X 0,Y 546.277,Z 396.122,A -85,B 0,C 180,E1 17487.586,E2 17487.586} C_VEL
LIN {X 0,Y 537.594,Z 385.376,A -85,B 0,C 180,E1 17485.622,E2 17485.622} C_VEL
LIN {X 0,Y 533.151,Z 380.052,A -85,B 0,C 180,E1 17484.545,E2 17484.545} C_VEL
LIN {X 0,Y 528.301,Z 374.273,A -85,B 0,C 180,E1 17483.301,E2 17483.301} C_VEL
LIN {X 0,Y 524.406,Z 369.552,A -85,B 0,C 180,E1 17482.24,E2 17482.24} C_VEL
LIN {X 0,Y 519.658,Z 364.41,A -85,B 0,C 180,E1 17480.882,E2 17480.882} C_VEL
LIN {X 0,Y 518.475,Z 362.662,A -85,B 0,C 180,E1 17480.405,E2 17480.405} C_VEL
LIN {X 0,Y 516.136,Z 358.764,A -85,B 0,C 180,E1 17478.994,E2 17478.994} C_VEL
LIN {X 0,Y 515.103,Z 357.042,A -85,B 0,C 180,E1 17478.329,E2 17478.329} C_VEL
LIN {X 0,Y 512.865,Z 353.198,A -85,B 0,C 180,E1 17476.771,E2 17476.771} C_VEL
LIN {X 0,Y 511.733,Z 351.55,A -85,B 0,C 180,E1 17475.992,E2 17475.992} C_VEL
LIN {X 0,Y 509.727,Z 348.307,A -85,B 0,C 180,E1 17474.426,E2 17474.426} C_VEL
LIN {X 0,Y 508.906,Z 346.622,A -85,B 0,C 180,E1 17473.637,E2 17473.637} C_VEL
LIN {X 0,Y 506.105,Z 342.467,A -85,B 0,C 180,E1 17471.048,E2 17471.048} C_VEL
LIN {X 0,Y 505.883,Z 341.314,A -85,B 0,C 180,E1 17470.247,E2 17470.247} C_VEL
LIN {X 0,Y 505.838,Z 341.138,A -85,B 0,C 180,E1 17466.697,E2 17466.697} C_VEL
LIN {X 0,Y 505.847,Z 341.216,A -85,B 0,C 180,E1 17463.173,E2 17463.173} C_VEL
LIN {X 0,Y 505.861,Z 341.131,A -85,B 0,C 180,E1 17459.66,E2 17459.66} C_VEL
LIN {X 0,Y 505.861,Z 341.196,A -85,B 0,C 180,E1 17456.147,E2 17456.147} C_VEL
LIN {X 0,Y 505.847,Z 341.138,A -85,B 0,C 180,E1 17452.618,E2 17452.618} C_VEL
LIN {X 0,Y 505.859,Z 341.161,A -85,B 0,C 180,E1 17449.177,E2 17449.177} C_VEL
LIN {X 0,Y 505.93,Z 341.662,A -85,B 0,C 180,E1 17447.676,E2 17447.676} C_VEL
LIN {X 0,Y 508.018,Z 345.722,A -85,B 0,C 180,E1 17445.292,E2 17445.292} C_VEL
LIN {X 0,Y 509.439,Z 347.543,A -85,B 0,C 180,E1 17444.168,E2 17444.168} C_VEL
LIN {X 0,Y 511.398,Z 351.196,A -85,B 0,C 180,E1 17442.476,E2 17442.476} C_VEL
LIN {X 0,Y 512.737,Z 352.953,A -85,B 0,C 180,E1 17441.584,E2 17441.584} C_VEL
LIN {X 0,Y 514.875,Z 356.884,A -85,B 0,C 180,E1 17440.014,E2 17440.014} C_VEL
LIN {X 0,Y 515.946,Z 358.503,A -85,B 0,C 180,E1 17439.347,E2 17439.347} C_VEL
LIN {X 0,Y 518.24,Z 362.478,A -85,B 0,C 180,E1 17437.899,E2 17437.899} C_VEL
LIN {X 0,Y 521.835,Z 368.909,A -85,B 0,C 180,E1 17435.791,E2 17435.791} C_VEL
LIN {X 0,Y 524.648,Z 374.148,A -85,B 0,C 180,E1 17434.244,E2 17434.244} C_VEL
LIN {X 0,Y 527.427,Z 379.33,A -85,B 0,C 180,E1 17432.814,E2 17432.814} C_VEL
LIN {X 0,Y 530.216,Z 384.39,A -85,B 0,C 180,E1 17431.534,E2 17431.534} C_VEL
LIN {X 0,Y 537.618,Z 394.128,A -85,B 0,C 180,E1 17429.703,E2 17429.703} C_VEL
LIN {X 0,Y 547.813,Z 407.82,A -85,B 0,C 180,E1 17427.422,E2 17427.422} C_VEL
LIN {X 0,Y 559.373,Z 424.366,A -85,B 0,C 180,E1 17425.078,E2 17425.078} C_VEL
LIN {X 0,Y 570.892,Z 441.817,A -85,B 0,C 180,E1 17422.951,E2 17422.951} C_VEL
LIN {X 0,Y 576.064,Z 450.483,A -85,B 0,C 180,E1 17422.041,E2 17422.041} C_VEL
LIN {X 0,Y 577.315,Z 458.89,A -85,B 0,C 180,E1 17421.699,E2 17421.699} C_VEL
LIN {X 0,Y 568.508,Z 689.883,A -85,B 0,C 180,E1 17418.365,E2 17418.365} C_VEL
LIN {X 0,Y 563.361,Z 831.083,A -85,B 0,C 180,E1 17416.34,E2 17416.34} C_VEL
LIN {X 0,Y 561.442,Z 857.5,A -85,B 0,C 180,E1 17415.834,E2 17415.834} C_VEL
LIN {X 0,Y 558.939,Z 881.483,A -85,B 0,C 180,E1 17415.199,E2 17415.199} C_VEL
LIN {X 0,Y 556.502,Z 901.041,A -85,B 0,C 180,E1 17414.557,E2 17414.557} C_VEL
LIN {X 0,Y 553.786,Z 919.924,A -85,B 0,C 180,E1 17413.822,E2 17413.822} C_VEL
LIN {X 0,Y 553.301,Z 923.248,A -85,B 0,C 180,E1 17413.683,E2 17413.683} C_VEL
LIN {X 0,Y 551.481,Z 930.436,A -85,B 0,C 180,E1 17413.441,E2 17413.441} C_VEL
LIN {X 0,Y 543.957,Z 948.656,A -85,B 0,C 180,E1 17412.993,E2 17412.993} C_VEL
LIN {X 0,Y 541.93,Z 955.519,A -85,B 0,C 180,E1 17412.696,E2 17412.696} C_VEL
LIN {X 0,Y 536.914,Z 980.305,A -85,B 0,C 180,E1 17411.179,E2 17411.179} C_VEL
LIN {X 0,Y 532.673,Z 999.493,A -85,B 0,C 180,E1 17409.799,E2 17409.799} C_VEL
LIN {X 0,Y 528.416,Z 1017.844,A -85,B 0,C 180,E1 17408.295,E2 17408.295} C_VEL
LIN {X 0,Y 523.083,Z 1039.852,A -85,B 0,C 180,E1 17406.204,E2 17406.204} C_VEL
LIN {X 0,Y 519.118,Z 1055.669,A -85,B 0,C 180,E1 17404.473,E2 17404.473} C_VEL
LIN {X 0,Y 515.352,Z 1070.583,A -85,B 0,C 180,E1 17402.641,E2 17402.641} C_VEL
LIN {X 0,Y 511.186,Z 1087.377,A -85,B 0,C 180,E1 17400.308,E2 17400.308} C_VEL
LIN {X 0,Y 507.455,Z 1102.602,A -85,B 0,C 180,E1 17397.839,E2 17397.839} C_VEL
LIN {X 0,Y 504.701,Z 1114.499,A -85,B 0,C 180,E1 17395.653,E2 17395.653} C_VEL
LIN {X 0,Y 501.982,Z 1127.3,A -85,B 0,C 180,E1 17392.98,E2 17392.98} C_VEL
LIN {X 0,Y 499.741,Z 1138.761,A -85,B 0,C 180,E1 17390.129,E2 17390.129} C_VEL
LIN {X 0,Y 498.303,Z 1147.516,A -85,B 0,C 180,E1 17387.61,E2 17387.61} C_VEL
LIN {X 0,Y 497.133,Z 1156.462,A -85,B 0,C 180,E1 17384.561,E2 17384.561} C_VEL
LIN {X 0,Y 496.477,Z 1162.918,A -85,B 0,C 180,E1 17381.82,E2 17381.82} C_VEL
LIN {X 0,Y 496.167,Z 1167.534,A -85,B 0,C 180,E1 17379.395,E2 17379.395} C_VEL
LIN {X 0,Y 495.985,Z 1171.445,A -85,B 0,C 180,E1 17376.715,E2 17376.715} C_VEL
LIN {X 0,Y 495.918,Z 1174.249,A -85,B 0,C 180,E1 17373.699,E2 17373.699} C_VEL
LIN {X 0,Y 495.918,Z 1175.346,A -85,B 0,C 180,E1 17371.156,E2 17371.156} C_VEL
LIN {X 0,Y 495.919,Z 1175.363,A -85,B 0,C 180,E1 17368.845,E2 17368.845} C_VEL
LIN {X 0,Y 495.911,Z 1174.367,A -85,B 0,C 180,E1 17366.417,E2 17366.417} C_VEL
LIN {X 0,Y 495.985,Z 1171.876,A -85,B 0,C 180,E1 17363.518,E2 17363.518} C_VEL
LIN {X 0,Y 496.158,Z 1167.683,A -85,B 0,C 180,E1 17360.606,E2 17360.606} C_VEL
LIN {X 0,Y 496.468,Z 1163.031,A -85,B 0,C 180,E1 17358.146,E2 17358.146} C_VEL
LIN {X 0,Y 497.105,Z 1156.686,A -85,B 0,C 180,E1 17355.438,E2 17355.438} C_VEL
LIN {X 0,Y 498.272,Z 1147.713,A -85,B 0,C 180,E1 17352.362,E2 17352.362} C_VEL
LIN {X 0,Y 499.678,Z 1139.077,A -85,B 0,C 180,E1 17349.869,E2 17349.869} C_VEL
LIN {X 0,Y 501.685,Z 1128.655,A -85,B 0,C 180,E1 17347.254,E2 17347.254} C_VEL
LIN {X 0,Y 504.549,Z 1115.151,A -85,B 0,C 180,E1 17344.383,E2 17344.383} C_VEL
LIN {X 0,Y 507.343,Z 1103.087,A -85,B 0,C 180,E1 17342.155,E2 17342.155} C_VEL
LIN {X 0,Y 510.853,Z 1088.656,A -85,B 0,C 180,E1 17339.8,E2 17339.8} C_VEL
LIN {X 0,Y 515.201,Z 1071.215,A -85,B 0,C 180,E1 17337.349,E2 17337.349} C_VEL
LIN {X 0,Y 519.059,Z 1055.933,A -85,B 0,C 180,E1 17335.465,E2 17335.465} C_VEL
LIN {X 0,Y 523.178,Z 1039.518,A -85,B 0,C 180,E1 17333.669,E2 17333.669} C_VEL
LIN {X 0,Y 528.376,Z 1018.094,A -85,B 0,C 180,E1 17331.634,E2 17331.634} C_VEL
LIN {X 0,Y 532.636,Z 999.758,A -85,B 0,C 180,E1 17330.129,E2 17330.129} C_VEL
LIN {X 0,Y 536.856,Z 980.664,A -85,B 0,C 180,E1 17328.753,E2 17328.753} C_VEL
LIN {X 0,Y 541.879,Z 955.911,A -85,B 0,C 180,E1 17327.232,E2 17327.232} C_VEL
LIN {X 0,Y 545.651,Z 935.169,A -85,B 0,C 180,E1 17326.159,E2 17326.159} C_VEL
LIN {X 0,Y 549.07,Z 914.223,A -85,B 0,C 180,E1 17325.234,E2 17325.234} C_VEL
LIN {X 0,Y 552.877,Z 886.784,A -85,B 0,C 180,E1 17324.252,E2 17324.252} C_VEL
LIN {X 0,Y 555.345,Z 864.707,A -85,B 0,C 180,E1 17323.633,E2 17323.633} C_VEL
LIN {X 0,Y 557.416,Z 841.646,A -85,B 0,C 180,E1 17323.132,E2 17323.132} C_VEL
LIN {X 0,Y 559.161,Z 807.277,A -85,B 0,C 180,E1 17322.592,E2 17322.592} C_VEL
LIN {X 0,Y 567.84,Z 576.349,A -85,B 0,C 180,E1 17319.271,E2 17319.271} C_VEL
LIN {X 0,Y 572.531,Z 459.682,A -85,B 0,C 180,E1 17317.554,E2 17317.554} C_VEL
LIN {X 0,Y 571.567,Z 454.64,A -85,B 0,C 180,E1 17317.313,E2 17317.313} C_VEL
LIN {X 0,Y 560.954,Z 437.911,A -85,B 0,C 180,E1 17315.371,E2 17315.371} C_VEL
LIN {X 0,Y 550.057,Z 421.723,A -85,B 0,C 180,E1 17313.203,E2 17313.203} C_VEL
LIN {X 0,Y 539.896,Z 407.523,A -85,B 0,C 180,E1 17310.988,E2 17310.988} C_VEL
LIN {X 0,Y 532.389,Z 397.525,A -85,B 0,C 180,E1 17309.199,E2 17309.199} C_VEL
LIN {X 0,Y 525.421,Z 388.456,A -85,B 0,C 180,E1 17307.391,E2 17307.391} C_VEL
LIN {X 0,Y 521.07,Z 382.719,A -85,B 0,C 180,E1 17306.129,E2 17306.129} C_VEL
LIN {X 0,Y 518.462,Z 377.924,A -85,B 0,C 180,E1 17304.74,E2 17304.74} C_VEL
LIN {X 0,Y 516.154,Z 373.572,A -85,B 0,C 180,E1 17303.399,E2 17303.399} C_VEL
LIN {X 0,Y 513.59,Z 368.904,A -85,B 0,C 180,E1 17301.83,E2 17301.83} C_VEL
LIN {X 0,Y 511.341,Z 364.942,A -85,B 0,C 180,E1 17300.369,E2 17300.369} C_VEL
LIN {X 0,Y 508.197,Z 359.427,A -85,B 0,C 180,E1 17298.112,E2 17298.112} C_VEL
LIN {X 0,Y 505.167,Z 354.631,A -85,B 0,C 180,E1 17295.734,E2 17295.734} C_VEL
LIN {X 0,Y 504.477,Z 353.235,A -85,B 0,C 180,E1 17295.049,E2 17295.049} C_VEL
LIN {X 0,Y 501.772,Z 349.095,A -85,B 0,C 180,E1 17292.428,E2 17292.428} C_VEL
LIN {X 0,Y 500.954,Z 347.555,A -85,B 0,C 180,E1 17291.397,E2 17291.397} C_VEL
LIN {X 0,Y 497.95,Z 342.402,A -85,B 0,C 180,E1 17286.051,E2 17286.051} C_VEL
LIN {X 0,Y 497.921,Z 342.165,A -85,B 0,C 180,E1 17282.417,E2 17282.417} C_VEL
LIN {X 0,Y 497.903,Z 342.133,A -85,B 0,C 180,E1 17278.964,E2 17278.964} C_VEL
LIN {X 0,Y 497.957,Z 342.475,A -85,B 0,C 180,E1 17275.393,E2 17275.393} C_VEL
LIN {X 0,Y 501.584,Z 348.421,A -85,B 0,C 180,E1 17269.548,E2 17269.548} C_VEL
LIN {X 0,Y 503.891,Z 352.624,A -85,B 0,C 180,E1 17267.042,E2 17267.042} C_VEL
LIN {X 0,Y 505.146,Z 354.285,A -85,B 0,C 180,E1 17266.026,E2 17266.026} C_VEL
LIN {X 0,Y 506.906,Z 357.752,A -85,B 0,C 180,E1 17264.439,E2 17264.439} C_VEL
LIN {X 0,Y 508.285,Z 359.386,A -85,B 0,C 180,E1 17263.544,E2 17263.544} C_VEL
LIN {X 0,Y 510.378,Z 363.334,A -85,B 0,C 180,E1 17261.968,E2 17261.968} C_VEL
LIN {X 0,Y 511.79,Z 365.095,A -85,B 0,C 180,E1 17261.312,E2 17261.312} C_VEL
LIN {X 0,Y 515.466,Z 369.431,A -85,B 0,C 180,E1 17260.097,E2 17260.097} C_VEL
LIN {X 0,Y 517.42,Z 371.456,A -85,B 0,C 180,E1 17259.497,E2 17259.497} C_VEL
LIN {X 0,Y 521.344,Z 375.916,A -85,B 0,C 180,E1 17258.334,E2 17258.334} C_VEL
LIN {X 0,Y 526.863,Z 382.244,A -85,B 0,C 180,E1 17256.809,E2 17256.809} C_VEL
LIN {X 0,Y 531.676,Z 388.067,A -85,B 0,C 180,E1 17255.56,E2 17255.56} C_VEL
LIN {X 0,Y 541.693,Z 400.595,A -85,B 0,C 180,E1 17253.172,E2 17253.172} C_VEL
LIN {X 0,Y 552.569,Z 414.743,A -85,B 0,C 180,E1 17250.842,E2 17250.842} C_VEL
LIN {X 0,Y 563.388,Z 429.836,A -85,B 0,C 180,E1 17248.726,E2 17248.726} C_VEL
LIN {X 0,Y 574.033,Z 445.327,A -85,B 0,C 180,E1 17246.812,E2 17246.812} C_VEL
LIN {X 0,Y 576.566,Z 449.687,A -85,B 0,C 180,E1 17246.366,E2 17246.366} C_VEL
LIN {X 0,Y 567.395,Z 659.725,A -85,B 0,C 180,E1 17243.172,E2 17243.172} C_VEL
LIN {X 0,Y 560.31,Z 826.384,A -85,B 0,C 180,E1 17240.644,E2 17240.644} C_VEL
LIN {X 0,Y 558.206,Z 853.534,A -85,B 0,C 180,E1 17240.12,E2 17240.12} C_VEL
LIN {X 0,Y 555.294,Z 880.119,A -85,B 0,C 180,E1 17239.412,E2 17239.412} C_VEL
LIN {X 0,Y 552.555,Z 901.363,A -85,B 0,C 180,E1 17238.713,E2 17238.713} C_VEL
LIN {X 0,Y 549.512,Z 922.216,A -85,B 0,C 180,E1 17237.896,E2 17237.896} C_VEL
LIN {X 0,Y 545.902,Z 944.419,A -85,B 0,C 180,E1 17236.877,E2 17236.877} C_VEL
LIN {X 0,Y 541.062,Z 970.955,A -85,B 0,C 180,E1 17235.43,E2 17235.43} C_VEL
LIN {X 0,Y 537.019,Z 991.338,A -85,B 0,C 180,E1 17234.135,E2 17234.135} C_VEL
LIN {X 0,Y 533.042,Z 1010.356,A -85,B 0,C 180,E1 17232.768,E2 17232.768} C_VEL
LIN {X 0,Y 528.182,Z 1033.076,A -85,B 0,C 180,E1 17230.919,E2 17230.919} C_VEL
LIN {X 0,Y 523.246,Z 1055.094,A -85,B 0,C 180,E1 17228.848,E2 17228.848} C_VEL
LIN {X 0,Y 519.539,Z 1071.565,A -85,B 0,C 180,E1 17227.11,E2 17227.11} C_VEL
LIN {X 0,Y 516.171,Z 1086.492,A -85,B 0,C 180,E1 17225.36,E2 17225.36} C_VEL
LIN {X 0,Y 512.716,Z 1101.841,A -85,B 0,C 180,E1 17223.363,E2 17223.363} C_VEL
LIN {X 0,Y 508.899,Z 1119.013,A -85,B 0,C 180,E1 17220.837,E2 17220.837} C_VEL
LIN {X 0,Y 505.753,Z 1133.787,A -85,B 0,C 180,E1 17218.325,E2 17218.325} C_VEL
LIN {X 0,Y 503.332,Z 1145.75,A -85,B 0,C 180,E1 17216.041,E2 17216.041} C_VEL
LIN {X 0,Y 501.606,Z 1154.89,A -85,B 0,C 180,E1 17214.081,E2 17214.081} C_VEL
LIN {X 0,Y 499.879,Z 1164.512,A -85,B 0,C 180,E1 17211.718,E2 17211.718} C_VEL
LIN {X 0,Y 498.545,Z 1173.1,A -85,B 0,C 180,E1 17209.324,E2 17209.324} C_VEL
LIN {X 0,Y 497.418,Z 1181.621,A -85,B 0,C 180,E1 17206.585,E2 17206.585} C_VEL
LIN {X 0,Y 496.6,Z 1189.79,A -85,B 0,C 180,E1 17203.388,E2 17203.388} C_VEL
LIN {X 0,Y 496.197,Z 1195.274,A -85,B 0,C 180,E1 17200.683,E2 17200.683} C_VEL
LIN {X 0,Y 496.018,Z 1199.233,A -85,B 0,C 180,E1 17198.199,E2 17198.199} C_VEL
LIN {X 0,Y 495.94,Z 1202.081,A -85,B 0,C 180,E1 17195.785,E2 17195.785} C_VEL
LIN {X 0,Y 495.915,Z 1203.959,A -85,B 0,C 180,E1 17193.352,E2 17193.352} C_VEL
LIN {X 0,Y 495.906,Z 1204.826,A -85,B 0,C 180,E1 17190.924,E2 17190.924} C_VEL
LIN {X 0,Y 495.91,Z 1204.712,A -85,B 0,C 180,E1 17188.498,E2 17188.498} C_VEL
LIN {X 0,Y 495.919,Z 1203.413,A -85,B 0,C 180,E1 17185.722,E2 17185.722} C_VEL
LIN {X 0,Y 495.989,Z 1200.309,A -85,B 0,C 180,E1 17182.587,E2 17182.587} C_VEL
LIN {X 0,Y 496.143,Z 1196.306,A -85,B 0,C 180,E1 17179.902,E2 17179.902} C_VEL
LIN {X 0,Y 496.455,Z 1191.314,A -85,B 0,C 180,E1 17177.318,E2 17177.318} C_VEL
LIN {X 0,Y 497.002,Z 1185.443,A -85,B 0,C 180,E1 17174.839,E2 17174.839} C_VEL
LIN {X 0,Y 497.897,Z 1177.732,A -85,B 0,C 180,E1 17172.106,E2 17172.106} C_VEL
LIN {X 0,Y 499.523,Z 1166.782,A -85,B 0,C 180,E1 17168.874,E2 17168.874} C_VEL
LIN {X 0,Y 501.325,Z 1156.416,A -85,B 0,C 180,E1 17166.274,E2 17166.274} C_VEL
LIN {X 0,Y 502.992,Z 1147.535,A -85,B 0,C 180,E1 17164.319,E2 17164.319} C_VEL
LIN {X 0,Y 505.329,Z 1135.77,A -85,B 0,C 180,E1 17162.034,E2 17162.034} C_VEL
LIN {X 0,Y 507.971,Z 1123.305,A -85,B 0,C 180,E1 17159.872,E2 17159.872} C_VEL
LIN {X 0,Y 511.191,Z 1108.615,A -85,B 0,C 180,E1 17157.592,E2 17157.592} C_VEL
LIN {X 0,Y 515.674,Z 1088.716,A -85,B 0,C 180,E1 17154.911,E2 17154.911} C_VEL
LIN {X 0,Y 519.421,Z 1072.111,A -85,B 0,C 180,E1 17152.949,E2 17152.949} C_VEL
LIN {X 0,Y 523.248,Z 1055.094,A -85,B 0,C 180,E1 17151.151,E2 17151.151} C_VEL
LIN {X 0,Y 528.181,Z 1033.066,A -85,B 0,C 180,E1 17149.08,E2 17149.08} C_VEL
LIN {X 0,Y 533.041,Z 1010.337,A -85,B 0,C 180,E1 17147.231,E2 17147.231} C_VEL
LIN {X 0,Y 537.018,Z 991.316,A -85,B 0,C 180,E1 17145.865,E2 17145.865} C_VEL
LIN {X 0,Y 541.242,Z 970.013,A -85,B 0,C 180,E1 17144.513,E2 17144.513} C_VEL
LIN {X 0,Y 546.082,Z 943.233,A -85,B 0,C 180,E1 17143.066,E2 17143.066} C_VEL
LIN {X 0,Y 549.609,Z 921.513,A -85,B 0,C 180,E1 17142.076,E2 17142.076} C_VEL
LIN {X 0,Y 552.657,Z 900.549,A -85,B 0,C 180,E1 17141.259,E2 17141.259} C_VEL
LIN {X 0,Y 555.531,Z 878.092,A -85,B 0,C 180,E1 17140.528,E2 17140.528} C_VEL
LIN {X 0,Y 558.548,Z 849.085,A -85,B 0,C 180,E1 17139.788,E2 17139.788} C_VEL
LIN {X 0,Y 560.358,Z 825.238,A -85,B 0,C 180,E1 17139.339,E2 17139.339} C_VEL
LIN {X 0,Y 569.185,Z 617.287,A -85,B 0,C 180,E1 17136.187,E2 17136.187} C_VEL
LIN {X 0,Y 576.504,Z 449.266,A -85,B 0,C 180,E1 17133.625,E2 17133.625} C_VEL
LIN {X 0,Y 564.901,Z 431.987,A -85,B 0,C 180,E1 17131.567,E2 17131.567} C_VEL
LIN {X 0,Y 553.635,Z 416.26,A -85,B 0,C 180,E1 17129.393,E2 17129.393} C_VEL
LIN {X 0,Y 543.535,Z 402.985,A -85,B 0,C 180,E1 17127.262,E2 17127.262} C_VEL
LIN {X 0,Y 534.958,Z 392.271,A -85,B 0,C 180,E1 17125.283,E2 17125.283} C_VEL
LIN {X 0,Y 530.869,Z 387.295,A -85,B 0,C 180,E1 17124.272,E2 17124.272} C_VEL
LIN {X 0,Y 525.977,Z 381.441,A -85,B 0,C 180,E1 17122.996,E2 17122.996} C_VEL
LIN {X 0,Y 521.223,Z 375.812,A -85,B 0,C 180,E1 17121.672,E2 17121.672} C_VEL
LIN {X 0,Y 517.3,Z 371.281,A -85,B 0,C 180,E1 17120.508,E2 17120.508} C_VEL
LIN {X 0,Y 512.013,Z 365.468,A -85,B 0,C 180,E1 17118.827,E2 17118.827} C_VEL
LIN {X 0,Y 510.916,Z 363.934,A -85,B 0,C 180,E1 17118.366,E2 17118.366} C_VEL
LIN {X 0,Y 508.429,Z 359.874,A -85,B 0,C 180,E1 17116.686,E2 17116.686} C_VEL
LIN {X 0,Y 507.511,Z 358.375,A -85,B 0,C 180,E1 17116.011,E2 17116.011} C_VEL
LIN {X 0,Y 505.435,Z 355.241,A -85,B 0,C 180,E1 17114.434,E2 17114.434} C_VEL
LIN {X 0,Y 504.689,Z 353.425,A -85,B 0,C 180,E1 17113.637,E2 17113.637} C_VEL
LIN {X 0,Y 501.771,Z 349.084,A -85,B 0,C 180,E1 17110.913,E2 17110.913} C_VEL
LIN {X 0,Y 501.05,Z 347.644,A -85,B 0,C 180,E1 17109.998,E2 17109.998} C_VEL
LIN {X 0,Y 497.932,Z 342.368,A -85,B 0,C 180,E1 17104.723,E2 17104.723} C_VEL
LIN {X 0,Y 497.902,Z 342.137,A -85,B 0,C 180,E1 17101.151,E2 17101.151} C_VEL
LIN {X 0,Y 497.92,Z 342.158,A -85,B 0,C 180,E1 17097.698,E2 17097.698} C_VEL
LIN {X 0,Y 497.935,Z 342.263,A -85,B 0,C 180,E1 17094.122,E2 17094.122} C_VEL
LIN {X 0,Y 498.107,Z 343.155,A -85,B 0,C 180,E1 17092.585,E2 17092.585} C_VEL
LIN {X 0,Y 501.566,Z 348.463,A -85,B 0,C 180,E1 17087.684,E2 17087.684} C_VEL
LIN {X 0,Y 503.923,Z 352.674,A -85,B 0,C 180,E1 17085.169,E2 17085.169} C_VEL
LIN {X 0,Y 505.022,Z 354.197,A -85,B 0,C 180,E1 17084.262,E2 17084.262} C_VEL
LIN {X 0,Y 507.145,Z 358.014,A -85,B 0,C 180,E1 17082.443,E2 17082.443} C_VEL
LIN {X 0,Y 508.265,Z 359.629,A -85,B 0,C 180,E1 17081.653,E2 17081.653} C_VEL
LIN {X 0,Y 510.418,Z 363.509,A -85,B 0,C 180,E1 17080.071,E2 17080.071} C_VEL
LIN {X 0,Y 511.427,Z 365.227,A -85,B 0,C 180,E1 17079.395,E2 17079.395} C_VEL
LIN {X 0,Y 514.278,Z 370.132,A -85,B 0,C 180,E1 17077.6,E2 17077.6} C_VEL
LIN {X 0,Y 517.265,Z 375.684,A -85,B 0,C 180,E1 17075.807,E2 17075.807} C_VEL
LIN {X 0,Y 520.068,Z 380.942,A -85,B 0,C 180,E1 17074.246,E2 17074.246} C_VEL
LIN {X 0,Y 522.376,Z 384.384,A -85,B 0,C 180,E1 17073.329,E2 17073.329} C_VEL
LIN {X 0,Y 530.903,Z 395.59,A -85,B 0,C 180,E1 17071.051,E2 17071.051} C_VEL
LIN {X 0,Y 535.429,Z 401.615,A -85,B 0,C 180,E1 17069.937,E2 17069.937} C_VEL
LIN {X 0,Y 544.881,Z 414.406,A -85,B 0,C 180,E1 17067.786,E2 17067.786} C_VEL
LIN {X 0,Y 556.301,Z 430.959,A -85,B 0,C 180,E1 17065.422,E2 17065.422} C_VEL
LIN {X 0,Y 567.57,Z 448.242,A -85,B 0,C 180,E1 17063.297,E2 17063.297} C_VEL
LIN {X 0,Y 571.777,Z 455.387,A -85,B 0,C 180,E1 17062.54,E2 17062.54} C_VEL
LIN {X 0,Y 572.527,Z 461.041,A -85,B 0,C 180,E1 17062.317,E2 17062.317} C_VEL
LIN {X 0,Y 563.363,Z 691.792,A -85,B 0,C 180,E1 17058.967,E2 17058.967} C_VEL
LIN {X 0,Y 558.072,Z 831.031,A -85,B 0,C 180,E1 17056.958,E2 17056.958} C_VEL
LIN {X 0,Y 556.088,Z 857.525,A -85,B 0,C 180,E1 17056.448,E2 17056.448} C_VEL
LIN {X 0,Y 553.528,Z 881.289,A -85,B 0,C 180,E1 17055.818,E2 17055.818} C_VEL
LIN {X 0,Y 551.065,Z 900.458,A -85,B 0,C 180,E1 17055.19,E2 17055.19} C_VEL
LIN {X 0,Y 548.243,Z 919.433,A -85,B 0,C 180,E1 17054.454,E2 17054.454} C_VEL
LIN {X 0,Y 544.384,Z 942.612,A -85,B 0,C 180,E1 17053.388,E2 17053.388} C_VEL
LIN {X 0,Y 541.93,Z 955.519,A -85,B 0,C 180,E1 17052.696,E2 17052.696} C_VEL
LIN {X 0,Y 539.859,Z 962.427,A -85,B 0,C 180,E1 17052.383,E2 17052.383} C_VEL
LIN {X 0,Y 531.784,Z 979.925,A -85,B 0,C 180,E1 17051.742,E2 17051.742} C_VEL
LIN {X 0,Y 529.623,Z 986.397,A -85,B 0,C 180,E1 17051.367,E2 17051.367} C_VEL
LIN {X 0,Y 524.51,Z 1008.515,A -85,B 0,C 180,E1 17049.689,E2 17049.689} C_VEL
LIN {X 0,Y 519.744,Z 1027.584,A -85,B 0,C 180,E1 17047.997,E2 17047.997} C_VEL
LIN {X 0,Y 515.656,Z 1043.531,A -85,B 0,C 180,E1 17046.395,E2 17046.395} C_VEL
LIN {X 0,Y 511.385,Z 1059.904,A -85,B 0,C 180,E1 17044.543,E2 17044.543} C_VEL
LIN {X 0,Y 506.393,Z 1078.779,A -85,B 0,C 180,E1 17042.083,E2 17042.083} C_VEL
LIN {X 0,Y 502.695,Z 1092.991,A -85,B 0,C 180,E1 17039.95,E2 17039.95} C_VEL
LIN {X 0,Y 499.184,Z 1107.056,A -85,B 0,C 180,E1 17037.562,E2 17037.562} C_VEL
LIN {X 0,Y 495.721,Z 1121.626,A -85,B 0,C 180,E1 17034.678,E2 17034.678} C_VEL
LIN {X 0,Y 493.425,Z 1132.159,A -85,B 0,C 180,E1 17032.268,E2 17032.268} C_VEL
LIN {X 0,Y 491.489,Z 1142.261,A -85,B 0,C 180,E1 17029.614,E2 17029.614} C_VEL
LIN {X 0,Y 489.86,Z 1152.182,A -85,B 0,C 180,E1 17026.483,E2 17026.483} C_VEL
LIN {X 0,Y 488.963,Z 1159.143,A -85,B 0,C 180,E1 17023.843,E2 17023.843} C_VEL
LIN {X 0,Y 488.359,Z 1165.608,A -85,B 0,C 180,E1 17020.858,E2 17020.858} C_VEL
LIN {X 0,Y 488.061,Z 1170.325,A -85,B 0,C 180,E1 17017.89,E2 17017.89} C_VEL
LIN {X 0,Y 487.948,Z 1173.166,A -85,B 0,C 180,E1 17015.409,E2 17015.409} C_VEL
LIN {X 0,Y 487.921,Z 1174.963,A -85,B 0,C 180,E1 17012.937,E2 17012.937} C_VEL
LIN {X 0,Y 487.918,Z 1175.793,A -85,B 0,C 180,E1 17010.118,E2 17010.118} C_VEL
LIN {X 0,Y 487.922,Z 1175.079,A -85,B 0,C 180,E1 17007.181,E2 17007.181} C_VEL
LIN {X 0,Y 487.948,Z 1173.359,A -85,B 0,C 180,E1 17004.709,E2 17004.709} C_VEL
LIN {X 0,Y 488.032,Z 1170.751,A -85,B 0,C 180,E1 17002.347,E2 17002.347} C_VEL
LIN {X 0,Y 488.235,Z 1166.974,A -85,B 0,C 180,E1 16999.856,E2 16999.856} C_VEL
LIN {X 0,Y 488.775,Z 1161.036,A -85,B 0,C 180,E1 16996.846,E2 16996.846} C_VEL
LIN {X 0,Y 489.635,Z 1153.782,A -85,B 0,C 180,E1 16993.998,E2 16993.998} C_VEL
LIN {X 0,Y 490.795,Z 1146.169,A -85,B 0,C 180,E1 16991.47,E2 16991.47} C_VEL
LIN {X 0,Y 492.695,Z 1135.967,A -85,B 0,C 180,E1 16988.575,E2 16988.575} C_VEL
LIN {X 0,Y 495.123,Z 1124.231,A -85,B 0,C 180,E1 16985.799,E2 16985.799} C_VEL
LIN {X 0,Y 497.679,Z 1113.187,A -85,B 0,C 180,E1 16983.512,E2 16983.512} C_VEL
LIN {X 0,Y 501.104,Z 1099.397,A -85,B 0,C 180,E1 16980.996,E2 16980.996} C_VEL
LIN {X 0,Y 505.184,Z 1083.457,A -85,B 0,C 180,E1 16978.499,E2 16978.499} C_VEL
LIN {X 0,Y 508.996,Z 1068.913,A -85,B 0,C 180,E1 16976.496,E2 16976.496} C_VEL
LIN {X 0,Y 513.282,Z 1052.683,A -85,B 0,C 180,E1 16974.514,E2 16974.514} C_VEL
LIN {X 0,Y 518.644,Z 1031.963,A -85,B 0,C 180,E1 16972.329,E2 16972.329} C_VEL
LIN {X 0,Y 522.972,Z 1014.635,A -85,B 0,C 180,E1 16970.74,E2 16970.74} C_VEL
LIN {X 0,Y 527.476,Z 995.922,A -85,B 0,C 180,E1 16969.23,E2 16969.23} C_VEL
LIN {X 0,Y 532.832,Z 971.965,A -85,B 0,C 180,E1 16967.576,E2 16967.576} C_VEL
LIN {X 0,Y 536.783,Z 952.556,A -85,B 0,C 180,E1 16966.433,E2 16966.433} C_VEL
LIN {X 0,Y 540.311,Z 933.603,A -85,B 0,C 180,E1 16965.464,E2 16965.464} C_VEL
LIN {X 0,Y 544.422,Z 909.099,A -85,B 0,C 180,E1 16964.404,E2 16964.404} C_VEL
LIN {X 0,Y 547.709,Z 885.071,A -85,B 0,C 180,E1 16963.576,E2 16963.576} C_VEL
LIN {X 0,Y 550.15,Z 863.654,A -85,B 0,C 180,E1 16962.98,E2 16962.98} C_VEL
LIN {X 0,Y 552.473,Z 838.19,A -85,B 0,C 180,E1 16962.437,E2 16962.437} C_VEL
LIN {X 0,Y 554.348,Z 797.346,A -85,B 0,C 180,E1 16961.818,E2 16961.818} C_VEL
LIN {X 0,Y 563.266,Z 570.465,A -85,B 0,C 180,E1 16958.533,E2 16958.533} C_VEL
LIN {X 0,Y 567.816,Z 461.707,A -85,B 0,C 180,E1 16956.922,E2 16956.922} C_VEL
LIN {X 0,Y 567.244,Z 459.419,A -85,B 0,C 180,E1 16956.79,E2 16956.79} C_VEL
LIN {X 0,Y 555.277,Z 440.528,A -85,B 0,C 180,E1 16954.526,E2 16954.526} C_VEL
LIN {X 0,Y 544.869,Z 425.136,A -85,B 0,C 180,E1 16952.371,E2 16952.371} C_VEL
LIN {X 0,Y 534.471,Z 410.628,A -85,B 0,C 180,E1 16949.998,E2 16949.998} C_VEL
LIN {X 0,Y 527.04,Z 400.612,A -85,B 0,C 180,E1 16948.129,E2 16948.129} C_VEL
LIN {X 0,Y 522.148,Z 394.385,A -85,B 0,C 180,E1 16946.806,E2 16946.806} C_VEL
LIN {X 0,Y 518.481,Z 389.575,A -85,B 0,C 180,E1 16945.747,E2 16945.747} C_VEL
LIN {X 0,Y 512.24,Z 381.277,A -85,B 0,C 180,E1 16943.71,E2 16943.71} C_VEL
LIN {X 0,Y 508.694,Z 375.025,A -85,B 0,C 180,E1 16941.566,E2 16941.566} C_VEL
LIN {X 0,Y 506.025,Z 370.195,A -85,B 0,C 180,E1 16939.749,E2 16939.749} C_VEL
LIN {X 0,Y 503.735,Z 366.103,A -85,B 0,C 180,E1 16938.038,E2 16938.038} C_VEL
LIN {X 0,Y 500.667,Z 360.995,A -85,B 0,C 180,E1 16935.522,E2 16935.522} C_VEL
LIN {X 0,Y 499.771,Z 359.578,A -85,B 0,C 180,E1 16934.72,E2 16934.72} C_VEL
LIN {X 0,Y 497.292,Z 355.301,A -85,B 0,C 180,E1 16932.07,E2 16932.07} C_VEL
LIN {X 0,Y 495.838,Z 353.483,A -85,B 0,C 180,E1 16930.457,E2 16930.457} C_VEL
LIN {X 0,Y 493.499,Z 349.026,A -85,B 0,C 180,E1 16925.931,E2 16925.931} C_VEL
LIN {X 0,Y 492.299,Z 347.833,A -85,B 0,C 180,E1 16921.513,E2 16921.513} C_VEL
LIN {X 0,Y 492.755,Z 348.33,A -85,B 0,C 180,E1 16917.558,E2 16917.558} C_VEL
LIN {X 0,Y 493.759,Z 349.559,A -85,B 0,C 180,E1 16915.004,E2 16915.004} C_VEL
LIN {X 0,Y 497.336,Z 355.278,A -85,B 0,C 180,E1 16909.575,E2 16909.575} C_VEL
LIN {X 0,Y 499.814,Z 359.592,A -85,B 0,C 180,E1 16906.935,E2 16906.935} C_VEL
LIN {X 0,Y 500.767,Z 360.925,A -85,B 0,C 180,E1 16906.137,E2 16906.137} C_VEL
LIN {X 0,Y 502.678,Z 364.576,A -85,B 0,C 180,E1 16904.423,E2 16904.423} C_VEL
LIN {X 0,Y 504.28,Z 366.381,A -85,B 0,C 180,E1 16903.617,E2 16903.617} C_VEL
LIN {X 0,Y 507.813,Z 370.53,A -85,B 0,C 180,E1 16902.289,E2 16902.289} C_VEL
LIN {X 0,Y 509.91,Z 372.557,A -85,B 0,C 180,E1 16901.567,E2 16901.567} C_VEL
LIN {X 0,Y 513.817,Z 377.113,A -85,B 0,C 180,E1 16900.267,E2 16900.267} C_VEL
LIN {X 0,Y 515.572,Z 379.064,A -85,B 0,C 180,E1 16899.716,E2 16899.716} C_VEL
LIN {X 0,Y 519.83,Z 383.76,A -85,B 0,C 180,E1 16898.445,E2 16898.445} C_VEL
LIN {X 0,Y 524.165,Z 389.073,A -85,B 0,C 180,E1 16897.217,E2 16897.217} C_VEL
LIN {X 0,Y 531.149,Z 397.643,A -85,B 0,C 180,E1 16895.386,E2 16895.386} C_VEL
LIN {X 0,Y 538.999,Z 407.451,A -85,B 0,C 180,E1 16893.503,E2 16893.503} C_VEL
LIN {X 0,Y 549.747,Z 421.608,A -85,B 0,C 180,E1 16891.155,E2 16891.155} C_VEL
LIN {X 0,Y 560.452,Z 436.72,A -85,B 0,C 180,E1 16889.022,E2 16889.022} C_VEL
LIN {X 0,Y 570.996,Z 452.271,A -85,B 0,C 180,E1 16887.092,E2 16887.092} C_VEL
LIN {X 0,Y 571.721,Z 453.72,A -85,B 0,C 180,E1 16886.957,E2 16886.957} C_VEL
LIN {X 0,Y 562.189,Z 664.065,A -85,B 0,C 180,E1 16883.743,E2 16883.743} C_VEL
LIN {X 0,Y 555.024,Z 826.333,A -85,B 0,C 180,E1 16881.265,E2 16881.265} C_VEL
LIN {X 0,Y 552.858,Z 853.452,A -85,B 0,C 180,E1 16880.74,E2 16880.74} C_VEL
LIN {X 0,Y 549.849,Z 880.082,A -85,B 0,C 180,E1 16880.03,E2 16880.03} C_VEL
LIN {X 0,Y 547.045,Z 901.149,A -85,B 0,C 180,E1 16879.334,E2 16879.334} C_VEL
LIN {X 0,Y 543.895,Z 922.003,A -85,B 0,C 180,E1 16878.515,E2 16878.515} C_VEL
LIN {X 0,Y 540.056,Z 944.777,A -85,B 0,C 180,E1 16877.465,E2 16877.465} C_VEL
LIN {X 0,Y 535.226,Z 970.266,A -85,B 0,C 180,E1 16876.068,E2 16876.068} C_VEL
LIN {X 0,Y 531.02,Z 990.67,A -85,B 0,C 180,E1 16874.766,E2 16874.766} C_VEL
LIN {X 0,Y 526.826,Z 1009.953,A -85,B 0,C 180,E1 16873.371,E2 16873.371} C_VEL
LIN {X 0,Y 522.193,Z 1030.521,A -85,B 0,C 180,E1 16871.688,E2 16871.688} C_VEL
LIN {X 0,Y 516.835,Z 1053.415,A -85,B 0,C 180,E1 16869.53,E2 16869.53} C_VEL
LIN {X 0,Y 512.622,Z 1071.256,A -85,B 0,C 180,E1 16867.626,E2 16867.626} C_VEL
LIN {X 0,Y 508.945,Z 1086.914,A -85,B 0,C 180,E1 16865.767,E2 16865.767} C_VEL
LIN {X 0,Y 504.808,Z 1104.66,A -85,B 0,C 180,E1 16863.41,E2 16863.41} C_VEL
LIN {X 0,Y 500.95,Z 1121.308,A -85,B 0,C 180,E1 16860.861,E2 16860.861} C_VEL
LIN {X 0,Y 498.023,Z 1134.611,A -85,B 0,C 180,E1 16858.543,E2 16858.543} C_VEL
LIN {X 0,Y 495.642,Z 1145.882,A -85,B 0,C 180,E1 16856.347,E2 16856.347} C_VEL
LIN {X 0,Y 493.545,Z 1156.721,A -85,B 0,C 180,E1 16853.978,E2 16853.978} C_VEL
LIN {X 0,Y 491.76,Z 1166.805,A -85,B 0,C 180,E1 16851.468,E2 16851.468} C_VEL
LIN {X 0,Y 490.049,Z 1177.736,A -85,B 0,C 180,E1 16848.19,E2 16848.19} C_VEL
LIN {X 0,Y 489.087,Z 1185.442,A -85,B 0,C 180,E1 16845.412,E2 16845.412} C_VEL
LIN {X 0,Y 488.503,Z 1191.313,A -85,B 0,C 180,E1 16842.891,E2 16842.891} C_VEL
LIN {X 0,Y 488.174,Z 1196.097,A -85,B 0,C 180,E1 16840.384,E2 16840.384} C_VEL
LIN {X 0,Y 487.993,Z 1200.148,A -85,B 0,C 180,E1 16837.653,E2 16837.653} C_VEL
LIN {X 0,Y 487.92,Z 1203.343,A -85,B 0,C 180,E1 16834.466,E2 16834.466} C_VEL
LIN {X 0,Y 487.908,Z 1204.69,A -85,B 0,C 180,E1 16831.644,E2 16831.644} C_VEL
LIN {X 0,Y 487.902,Z 1204.848,A -85,B 0,C 180,E1 16829.178,E2 16829.178} C_VEL
LIN {X 0,Y 487.916,Z 1204.023,A -85,B 0,C 180,E1 16826.71,E2 16826.71} C_VEL
LIN {X 0,Y 487.939,Z 1202.19,A -85,B 0,C 180,E1 16824.237,E2 16824.237} C_VEL
LIN {X 0,Y 488.022,Z 1199.317,A -85,B 0,C 180,E1 16821.732,E2 16821.732} C_VEL
LIN {X 0,Y 488.207,Z 1195.476,A -85,B 0,C 180,E1 16819.259,E2 16819.259} C_VEL
LIN {X 0,Y 488.605,Z 1190.294,A -85,B 0,C 180,E1 16816.63,E2 16816.63} C_VEL
LIN {X 0,Y 489.408,Z 1182.676,A -85,B 0,C 180,E1 16813.502,E2 16813.502} C_VEL
LIN {X 0,Y 490.675,Z 1173.502,A -85,B 0,C 180,E1 16810.476,E2 16810.476} C_VEL
LIN {X 0,Y 492.079,Z 1164.964,A -85,B 0,C 180,E1 16808.045,E2 16808.045} C_VEL
LIN {X 0,Y 493.833,Z 1155.174,A -85,B 0,C 180,E1 16805.664,E2 16805.664} C_VEL
LIN {X 0,Y 496.072,Z 1143.903,A -85,B 0,C 180,E1 16803.243,E2 16803.243} C_VEL
LIN {X 0,Y 499.362,Z 1128.512,A -85,B 0,C 180,E1 16800.345,E2 16800.345} C_VEL
LIN {X 0,Y 502.742,Z 1113.541,A -85,B 0,C 180,E1 16797.915,E2 16797.915} C_VEL
LIN {X 0,Y 506.014,Z 1099.363,A -85,B 0,C 180,E1 16795.862,E2 16795.862} C_VEL
LIN {X 0,Y 509.617,Z 1084.025,A -85,B 0,C 180,E1 16793.872,E2 16793.872} C_VEL
LIN {X 0,Y 514.139,Z 1064.878,A -85,B 0,C 180,E1 16791.656,E2 16791.656} C_VEL
LIN {X 0,Y 519.096,Z 1043.755,A -85,B 0,C 180,E1 16789.524,E2 16789.524} C_VEL
LIN {X 0,Y 523.327,Z 1025.474,A -85,B 0,C 180,E1 16787.884,E2 16787.884} C_VEL
LIN {X 0,Y 527.562,Z 1006.653,A -85,B 0,C 180,E1 16786.379,E2 16786.379} C_VEL
LIN {X 0,Y 532.706,Z 982.992,A -85,B 0,C 180,E1 16784.718,E2 16784.718} C_VEL
LIN {X 0,Y 537.318,Z 959.449,A -85,B 0,C 180,E1 16783.314,E2 16783.314} C_VEL
LIN {X 0,Y 541.013,Z 939.088,A -85,B 0,C 180,E1 16782.26,E2 16782.26} C_VEL
LIN {X 0,Y 544.504,Z 918.023,A -85,B 0,C 180,E1 16781.318,E2 16781.318} C_VEL
LIN {X 0,Y 548.378,Z 891.904,A -85,B 0,C 180,E1 16780.338,E2 16780.338} C_VEL
LIN {X 0,Y 551.513,Z 865.601,A -85,B 0,C 180,E1 16779.566,E2 16779.566} C_VEL
LIN {X 0,Y 553.645,Z 844.049,A -85,B 0,C 180,E1 16779.067,E2 16779.067} C_VEL
LIN {X 0,Y 555.295,Z 821.387,A -85,B 0,C 180,E1 16778.655,E2 16778.655} C_VEL
LIN {X 0,Y 564.875,Z 603.087,A -85,B 0,C 180,E1 16775.331,E2 16775.331} C_VEL
LIN {X 0,Y 571.596,Z 453.247,A -85,B 0,C 180,E1 16773.024,E2 16773.024} C_VEL
LIN {X 0,Y 560.871,Z 437.367,A -85,B 0,C 180,E1 16771.072,E2 16771.072} C_VEL
LIN {X 0,Y 550.236,Z 422.348,A -85,B 0,C 180,E1 16768.966,E2 16768.966} C_VEL
LIN {X 0,Y 540.386,Z 409.315,A -85,B 0,C 180,E1 16766.839,E2 16766.839} C_VEL
LIN {X 0,Y 532.143,Z 398.919,A -85,B 0,C 180,E1 16764.891,E2 16764.891} C_VEL
LIN {X 0,Y 528.404,Z 394.33,A -85,B 0,C 180,E1 16763.947,E2 16763.947} C_VEL
LIN {X 0,Y 523.859,Z 388.789,A -85,B 0,C 180,E1 16762.738,E2 16762.738} C_VEL
LIN {X 0,Y 518.98,Z 383.012,A -85,B 0,C 180,E1 16761.355,E2 16761.355} C_VEL
LIN {X 0,Y 515.044,Z 378.276,A -85,B 0,C 180,E1 16760.157,E2 16760.157} C_VEL
LIN {X 0,Y 510.226,Z 373.051,A -85,B 0,C 180,E1 16758.599,E2 16758.599} C_VEL
LIN {X 0,Y 508.763,Z 371.312,A -85,B 0,C 180,E1 16758.091,E2 16758.091} C_VEL
LIN {X 0,Y 504.737,Z 367.091,A -85,B 0,C 180,E1 16756.634,E2 16756.634} C_VEL
LIN {X 0,Y 503.448,Z 365.34,A -85,B 0,C 180,E1 16756.085,E2 16756.085} C_VEL
LIN {X 0,Y 501.049,Z 361.881,A -85,B 0,C 180,E1 16754.327,E2 16754.327} C_VEL
LIN {X 0,Y 500.305,Z 360.082,A -85,B 0,C 180,E1 16753.523,E2 16753.523} C_VEL
LIN {X 0,Y 497.453,Z 355.71,A -85,B 0,C 180,E1 16750.774,E2 16750.774} C_VEL
LIN {X 0,Y 496.711,Z 354.333,A -85,B 0,C 180,E1 16749.852,E2 16749.852} C_VEL
LIN {X 0,Y 493.46,Z 348.961,A -85,B 0,C 180,E1 16744.533,E2 16744.533} C_VEL
LIN {X 0,Y 492.128,Z 347.639,A -85,B 0,C 180,E1 16740,E2 16740} C_VEL
LIN {X 0,Y 492.626,Z 348.188,A -85,B 0,C 180,E1 16735.693,E2 16735.693} C_VEL
LIN {X 0,Y 493.739,Z 349.52,A -85,B 0,C 180,E1 16733.021,E2 16733.021} C_VEL
LIN {X 0,Y 497.265,Z 355.211,A -85,B 0,C 180,E1 16727.75,E2 16727.75} C_VEL
LIN {X 0,Y 499.677,Z 359.475,A -85,B 0,C 180,E1 16725.159,E2 16725.159} C_VEL
LIN {X 0,Y 500.608,Z 360.847,A -85,B 0,C 180,E1 16724.357,E2 16724.357} C_VEL
LIN {X 0,Y 502.718,Z 364.643,A -85,B 0,C 180,E1 16722.522,E2 16722.522} C_VEL
LIN {X 0,Y 503.798,Z 366.31,A -85,B 0,C 180,E1 16721.725,E2 16721.725} C_VEL
LIN {X 0,Y 506.16,Z 370.365,A -85,B 0,C 180,E1 16720.016,E2 16720.016} C_VEL
LIN {X 0,Y 509.293,Z 375.736,A -85,B 0,C 180,E1 16717.976,E2 16717.976} C_VEL
LIN {X 0,Y 511.857,Z 380.472,A -85,B 0,C 180,E1 16716.393,E2 16716.393} C_VEL
LIN {X 0,Y 513.733,Z 383.705,A -85,B 0,C 180,E1 16715.569,E2 16715.569} C_VEL
LIN {X 0,Y 520.685,Z 392.386,A -85,B 0,C 180,E1 16713.482,E2 16713.482} C_VEL
LIN {X 0,Y 528.095,Z 402.055,A -85,B 0,C 180,E1 16711.471,E2 16711.471} C_VEL
LIN {X 0,Y 536.559,Z 413.425,A -85,B 0,C 180,E1 16709.389,E2 16709.389} C_VEL
LIN {X 0,Y 547.572,Z 429.071,A -85,B 0,C 180,E1 16706.939,E2 16706.939} C_VEL
LIN {X 0,Y 559.58,Z 447.219,A -85,B 0,C 180,E1 16704.529,E2 16704.529} C_VEL
LIN {X 0,Y 567.524,Z 460.191,A -85,B 0,C 180,E1 16703.05,E2 16703.05} C_VEL
LIN {X 0,Y 567.797,Z 463.393,A -85,B 0,C 180,E1 16702.942,E2 16702.942} C_VEL
LIN {X 0,Y 558.278,Z 693.723,A -85,B 0,C 180,E1 16699.581,E2 16699.581} C_VEL
LIN {X 0,Y 552.839,Z 831.108,A -85,B 0,C 180,E1 16697.585,E2 16697.585} C_VEL
LIN {X 0,Y 550.773,Z 857.741,A -85,B 0,C 180,E1 16697.069,E2 16697.069} C_VEL
LIN {X 0,Y 548.151,Z 881.329,A -85,B 0,C 180,E1 16696.442,E2 16696.442} C_VEL
LIN {X 0,Y 545.59,Z 900.594,A -85,B 0,C 180,E1 16695.81,E2 16695.81} C_VEL
LIN {X 0,Y 542.572,Z 920.197,A -85,B 0,C 180,E1 16695.044,E2 16695.044} C_VEL
LIN {X 0,Y 538.393,Z 944.329,A -85,B 0,C 180,E1 16693.92,E2 16693.92} C_VEL
LIN {X 0,Y 533.964,Z 966.37,A -85,B 0,C 180,E1 16692.677,E2 16692.677} C_VEL
LIN {X 0,Y 529.948,Z 984.894,A -85,B 0,C 180,E1 16691.472,E2 16691.472} C_VEL
LIN {X 0,Y 529.623,Z 986.397,A -85,B 0,C 180,E1 16691.367,E2 16691.367} C_VEL
LIN {X 0,Y 527.449,Z 992.973,A -85,B 0,C 180,E1 16690.976,E2 16690.976} C_VEL
LIN {X 0,Y 518.474,Z 1010.442,A -85,B 0,C 180,E1 16690.082,E2 16690.082} C_VEL
LIN {X 0,Y 516.537,Z 1015.623,A -85,B 0,C 180,E1 16689.69,E2 16689.69} C_VEL
LIN {X 0,Y 511.564,Z 1034.811,A -85,B 0,C 180,E1 16687.901,E2 16687.901} C_VEL
LIN {X 0,Y 506.237,Z 1054.383,A -85,B 0,C 180,E1 16685.777,E2 16685.777} C_VEL
LIN {X 0,Y 502.062,Z 1069.581,A -85,B 0,C 180,E1 16683.892,E2 16683.892} C_VEL
LIN {X 0,Y 498.093,Z 1084.085,A -85,B 0,C 180,E1 16681.867,E2 16681.867} C_VEL
LIN {X 0,Y 493.459,Z 1101.315,A -85,B 0,C 180,E1 16679.098,E2 16679.098} C_VEL
LIN {X 0,Y 490.25,Z 1113.725,A -85,B 0,C 180,E1 16676.791,E2 16676.791} C_VEL
LIN {X 0,Y 487.449,Z 1125.302,A -85,B 0,C 180,E1 16674.35,E2 16674.35} C_VEL
LIN {X 0,Y 484.609,Z 1138.251,A -85,B 0,C 180,E1 16671.154,E2 16671.154} C_VEL
LIN {X 0,Y 482.94,Z 1147.024,A -85,B 0,C 180,E1 16668.593,E2 16668.593} C_VEL
LIN {X 0,Y 481.682,Z 1154.913,A -85,B 0,C 180,E1 16665.903,E2 16665.903} C_VEL
LIN {X 0,Y 480.698,Z 1162.745,A -85,B 0,C 180,E1 16662.616,E2 16662.616} C_VEL
LIN {X 0,Y 480.245,Z 1167.719,A -85,B 0,C 180,E1 16659.951,E2 16659.951} C_VEL
LIN {X 0,Y 480.044,Z 1171.373,A -85,B 0,C 180,E1 16657.42,E2 16657.42} C_VEL
LIN {X 0,Y 479.937,Z 1174.413,A -85,B 0,C 180,E1 16654.421,E2 16654.421} C_VEL
LIN {X 0,Y 479.921,Z 1175.798,A -85,B 0,C 180,E1 16651.433,E2 16651.433} C_VEL
LIN {X 0,Y 479.925,Z 1175.88,A -85,B 0,C 180,E1 16648.926,E2 16648.926} C_VEL
LIN {X 0,Y 479.921,Z 1175.002,A -85,B 0,C 180,E1 16646.536,E2 16646.536} C_VEL
LIN {X 0,Y 479.976,Z 1172.961,A -85,B 0,C 180,E1 16643.902,E2 16643.902} C_VEL
LIN {X 0,Y 480.171,Z 1169.045,A -85,B 0,C 180,E1 16640.767,E2 16640.767} C_VEL
LIN {X 0,Y 480.548,Z 1164.139,A -85,B 0,C 180,E1 16637.991,E2 16637.991} C_VEL
LIN {X 0,Y 481.178,Z 1158.53,A -85,B 0,C 180,E1 16635.438,E2 16635.438} C_VEL
LIN {X 0,Y 482.349,Z 1150.66,A -85,B 0,C 180,E1 16632.471,E2 16632.471} C_VEL
LIN {X 0,Y 484.105,Z 1140.732,A -85,B 0,C 180,E1 16629.444,E2 16629.444} C_VEL
LIN {X 0,Y 486.066,Z 1131.373,A -85,B 0,C 180,E1 16626.993,E2 16626.993} C_VEL
LIN {X 0,Y 489.063,Z 1118.684,A -85,B 0,C 180,E1 16624.104,E2 16624.104} C_VEL
LIN {X 0,Y 492.451,Z 1105.183,A -85,B 0,C 180,E1 16621.501,E2 16621.501} C_VEL
LIN {X 0,Y 495.831,Z 1092.388,A -85,B 0,C 180,E1 16619.324,E2 16619.324} C_VEL
LIN {X 0,Y 500.398,Z 1075.886,A -85,B 0,C 180,E1 16616.85,E2 16616.85} C_VEL
LIN {X 0,Y 505.266,Z 1058.018,A -85,B 0,C 180,E1 16614.562,E2 16614.562} C_VEL
LIN {X 0,Y 509.484,Z 1042.516,A -85,B 0,C 180,E1 16612.81,E2 16612.81} C_VEL
LIN {X 0,Y 514.42,Z 1024.063,A -85,B 0,C 180,E1 16610.968,E2 16610.968} C_VEL
LIN {X 0,Y 519.761,Z 1002.881,A -85,B 0,C 180,E1 16609.151,E2 16609.151} C_VEL
LIN {X 0,Y 524.265,Z 983.997,A -85,B 0,C 180,E1 16607.749,E2 16607.749} C_VEL
LIN {X 0,Y 528.809,Z 963.654,A -85,B 0,C 180,E1 16606.434,E2 16606.434} C_VEL
LIN {X 0,Y 533.805,Z 938.715,A -85,B 0,C 180,E1 16605.076,E2 16605.076} C_VEL
LIN {X 0,Y 537.55,Z 917.504,A -85,B 0,C 180,E1 16604.112,E2 16604.112} C_VEL
LIN {X 0,Y 541.121,Z 894.526,A -85,B 0,C 180,E1 16603.24,E2 16603.24} C_VEL
LIN {X 0,Y 544.442,Z 867.97,A -85,B 0,C 180,E1 16602.449,E2 16602.449} C_VEL
LIN {X 0,Y 546.611,Z 846.059,A -85,B 0,C 180,E1 16601.953,E2 16601.953} C_VEL
LIN {X 0,Y 548.221,Z 822.292,A -85,B 0,C 180,E1 16601.54,E2 16601.54} C_VEL
LIN {X 0,Y 557.849,Z 586.551,A -85,B 0,C 180,E1 16598.108,E2 16598.108} C_VEL
LIN {X 0,Y 563.185,Z 464.575,A -85,B 0,C 180,E1 16596.3,E2 16596.3} C_VEL
LIN {X 0,Y 551.896,Z 446.638,A -85,B 0,C 180,E1 16594.111,E2 16594.111} C_VEL
LIN {X 0,Y 541.943,Z 431.739,A -85,B 0,C 180,E1 16592.004,E2 16592.004} C_VEL
LIN {X 0,Y 531.891,Z 417.532,A -85,B 0,C 180,E1 16589.662,E2 16589.662} C_VEL
LIN {X 0,Y 524.559,Z 407.524,A -85,B 0,C 180,E1 16587.779,E2 16587.779} C_VEL
LIN {X 0,Y 516.747,Z 397.253,A -85,B 0,C 180,E1 16585.563,E2 16585.563} C_VEL
LIN {X 0,Y 508.974,Z 387.355,A -85,B 0,C 180,E1 16583.074,E2 16583.074} C_VEL
LIN {X 0,Y 504.057,Z 381.274,A -85,B 0,C 180,E1 16581.286,E2 16581.286} C_VEL
LIN {X 0,Y 501.384,Z 376.596,A -85,B 0,C 180,E1 16579.575,E2 16579.575} C_VEL
LIN {X 0,Y 498.545,Z 371.544,A -85,B 0,C 180,E1 16577.388,E2 16577.388} C_VEL
LIN {X 0,Y 496.26,Z 367.643,A -85,B 0,C 180,E1 16575.424,E2 16575.424} C_VEL
LIN {X 0,Y 495.379,Z 366.223,A -85,B 0,C 180,E1 16574.614,E2 16574.614} C_VEL
LIN {X 0,Y 492.964,Z 361.934,A -85,B 0,C 180,E1 16571.94,E2 16571.94} C_VEL
LIN {X 0,Y 489.364,Z 355.891,A -85,B 0,C 180,E1 16565.981,E2 16565.981} C_VEL
LIN {X 0,Y 488.157,Z 354.677,A -85,B 0,C 180,E1 16561.526,E2 16561.526} C_VEL
LIN {X 0,Y 488.622,Z 355.183,A -85,B 0,C 180,E1 16557.537,E2 16557.537} C_VEL
LIN {X 0,Y 489.581,Z 356.351,A -85,B 0,C 180,E1 16555.079,E2 16555.079} C_VEL
LIN {X 0,Y 493.027,Z 361.901,A -85,B 0,C 180,E1 16549.719,E2 16549.719} C_VEL
LIN {X 0,Y 495.453,Z 366.243,A -85,B 0,C 180,E1 16547.055,E2 16547.055} C_VEL
LIN {X 0,Y 496.904,Z 367.86,A -85,B 0,C 180,E1 16546.264,E2 16546.264} C_VEL
LIN {X 0,Y 500.161,Z 371.745,A -85,B 0,C 180,E1 16544.818,E2 16544.818} C_VEL
LIN {X 0,Y 502.579,Z 373.933,A -85,B 0,C 180,E1 16543.857,E2 16543.857} C_VEL
LIN {X 0,Y 506.226,Z 378.207,A -85,B 0,C 180,E1 16542.469,E2 16542.469} C_VEL
LIN {X 0,Y 508.14,Z 380.139,A -85,B 0,C 180,E1 16541.797,E2 16541.797} C_VEL
LIN {X 0,Y 512.172,Z 384.794,A -85,B 0,C 180,E1 16540.439,E2 16540.439} C_VEL
LIN {X 0,Y 518.715,Z 392.497,A -85,B 0,C 180,E1 16538.426,E2 16538.426} C_VEL
LIN {X 0,Y 523.712,Z 398.549,A -85,B 0,C 180,E1 16537.018,E2 16537.018} C_VEL
LIN {X 0,Y 529.159,Z 405.275,A -85,B 0,C 180,E1 16535.585,E2 16535.585} C_VEL
LIN {X 0,Y 536.631,Z 414.733,A -85,B 0,C 180,E1 16533.764,E2 16533.764} C_VEL
LIN {X 0,Y 546.943,Z 428.471,A -85,B 0,C 180,E1 16531.471,E2 16531.471} C_VEL
LIN {X 0,Y 557.652,Z 443.769,A -85,B 0,C 180,E1 16529.298,E2 16529.298} C_VEL
LIN {X 0,Y 566.944,Z 457.654,A -85,B 0,C 180,E1 16527.56,E2 16527.56} C_VEL
LIN {X 0,Y 557.019,Z 668.875,A -85,B 0,C 180,E1 16524.317,E2 16524.317} C_VEL
LIN {X 0,Y 549.8,Z 826.431,A -85,B 0,C 180,E1 16521.896,E2 16521.896} C_VEL
LIN {X 0,Y 547.561,Z 853.596,A -85,B 0,C 180,E1 16521.368,E2 16521.368} C_VEL
LIN {X 0,Y 544.451,Z 880.228,A -85,B 0,C 180,E1 16520.655,E2 16520.655} C_VEL
LIN {X 0,Y 541.494,Z 901.714,A -85,B 0,C 180,E1 16519.94,E2 16519.94} C_VEL
LIN {X 0,Y 538.239,Z 922.475,A -85,B 0,C 180,E1 16519.119,E2 16519.119} C_VEL
LIN {X 0,Y 533.885,Z 947.468,A -85,B 0,C 180,E1 16517.951,E2 16517.951} C_VEL
LIN {X 0,Y 529.08,Z 971.456,A -85,B 0,C 180,E1 16516.605,E2 16516.605} C_VEL
LIN {X 0,Y 524.736,Z 991.711,A -85,B 0,C 180,E1 16515.295,E2 16515.295} C_VEL
LIN {X 0,Y 520.287,Z 1011.356,A -85,B 0,C 180,E1 16513.852,E2 16513.852} C_VEL
LIN {X 0,Y 514.867,Z 1034.393,A -85,B 0,C 180,E1 16511.917,E2 16511.917} C_VEL
LIN {X 0,Y 509.803,Z 1054.842,A -85,B 0,C 180,E1 16509.925,E2 16509.925} C_VEL
LIN {X 0,Y 505.616,Z 1071.662,A -85,B 0,C 180,E1 16508.087,E2 16508.087} C_VEL
LIN {X 0,Y 500.761,Z 1091.492,A -85,B 0,C 180,E1 16505.664,E2 16505.664} C_VEL
LIN {X 0,Y 496.467,Z 1108.891,A -85,B 0,C 180,E1 16503.216,E2 16503.216} C_VEL
LIN {X 0,Y 493.144,Z 1122.881,A -85,B 0,C 180,E1 16500.997,E2 16500.997} C_VEL
LIN {X 0,Y 490.3,Z 1135.432,A -85,B 0,C 180,E1 16498.769,E2 16498.769} C_VEL
LIN {X 0,Y 487.598,Z 1147.808,A -85,B 0,C 180,E1 16496.291,E2 16496.291} C_VEL
LIN {X 0,Y 484.867,Z 1161.724,A -85,B 0,C 180,E1 16493.067,E2 16493.067} C_VEL
LIN {X 0,Y 483.189,Z 1171.309,A -85,B 0,C 180,E1 16490.47,E2 16490.47} C_VEL
LIN {X 0,Y 482.073,Z 1178.582,A -85,B 0,C 180,E1 16488.201,E2 16488.201} C_VEL
LIN {X 0,Y 481.139,Z 1185.742,A -85,B 0,C 180,E1 16485.55,E2 16485.55} C_VEL
LIN {X 0,Y 480.53,Z 1191.564,A -85,B 0,C 180,E1 16482.986,E2 16482.986} C_VEL
LIN {X 0,Y 480.172,Z 1196.508,A -85,B 0,C 180,E1 16480.316,E2 16480.316} C_VEL
LIN {X 0,Y 479.98,Z 1200.927,A -85,B 0,C 180,E1 16477.18,E2 16477.18} C_VEL
LIN {X 0,Y 479.916,Z 1203.613,A -85,B 0,C 180,E1 16474.062,E2 16474.062} C_VEL
LIN {X 0,Y 479.911,Z 1204.735,A -85,B 0,C 180,E1 16471.432,E2 16471.432} C_VEL
LIN {X 0,Y 479.907,Z 1204.825,A -85,B 0,C 180,E1 16469.045,E2 16469.045} C_VEL
LIN {X 0,Y 479.915,Z 1203.952,A -85,B 0,C 180,E1 16466.536,E2 16466.536} C_VEL
LIN {X 0,Y 479.944,Z 1202.073,A -85,B 0,C 180,E1 16464.021,E2 16464.021} C_VEL
LIN {X 0,Y 480.037,Z 1199.185,A -85,B 0,C 180,E1 16461.495,E2 16461.495} C_VEL
LIN {X 0,Y 480.238,Z 1195.267,A -85,B 0,C 180,E1 16458.957,E2 16458.957} C_VEL
LIN {X 0,Y 480.712,Z 1189.782,A -85,B 0,C 180,E1 16456.16,E2 16456.16} C_VEL
LIN {X 0,Y 481.701,Z 1181.262,A -85,B 0,C 180,E1 16452.733,E2 16452.733} C_VEL
LIN {X 0,Y 482.8,Z 1173.817,A -85,B 0,C 180,E1 16450.271,E2 16450.271} C_VEL
LIN {X 0,Y 484.34,Z 1164.581,A -85,B 0,C 180,E1 16447.675,E2 16447.675} C_VEL
LIN {X 0,Y 486.233,Z 1154.499,A -85,B 0,C 180,E1 16445.197,E2 16445.197} C_VEL
LIN {X 0,Y 488.877,Z 1141.87,A -85,B 0,C 180,E1 16442.469,E2 16442.469} C_VEL
LIN {X 0,Y 492.495,Z 1125.821,A -85,B 0,C 180,E1 16439.499,E2 16439.499} C_VEL
LIN {X 0,Y 495.74,Z 1111.99,A -85,B 0,C 180,E1 16437.254,E2 16437.254} C_VEL
LIN {X 0,Y 499.167,Z 1097.746,A -85,B 0,C 180,E1 16435.188,E2 16435.188} C_VEL
LIN {X 0,Y 503.588,Z 1079.862,A -85,B 0,C 180,E1 16432.872,E2 16432.872} C_VEL
LIN {X 0,Y 508.751,Z 1059.113,A -85,B 0,C 180,E1 16430.521,E2 16430.521} C_VEL
LIN {X 0,Y 513.001,Z 1041.896,A -85,B 0,C 180,E1 16428.792,E2 16428.792} C_VEL
LIN {X 0,Y 517.195,Z 1024.521,A -85,B 0,C 180,E1 16427.228,E2 16427.228} C_VEL
LIN {X 0,Y 521.884,Z 1004.543,A -85,B 0,C 180,E1 16425.629,E2 16425.629} C_VEL
LIN {X 0,Y 527.388,Z 979.698,A -85,B 0,C 180,E1 16423.909,E2 16423.909} C_VEL
LIN {X 0,Y 531.646,Z 958.737,A -85,B 0,C 180,E1 16422.662,E2 16422.662} C_VEL
LIN {X 0,Y 535.492,Z 938.204,A -85,B 0,C 180,E1 16421.598,E2 16421.598} C_VEL
LIN {X 0,Y 539.217,Z 916.421,A -85,B 0,C 180,E1 16420.628,E2 16420.628} C_VEL
LIN {X 0,Y 543.403,Z 888.346,A -85,B 0,C 180,E1 16419.6,E2 16419.6} C_VEL
LIN {X 0,Y 546.285,Z 864.682,A -85,B 0,C 180,E1 16418.913,E2 16418.913} C_VEL
LIN {X 0,Y 548.46,Z 843.192,A -85,B 0,C 180,E1 16418.418,E2 16418.418} C_VEL
LIN {X 0,Y 550.19,Z 819.571,A -85,B 0,C 180,E1 16417.992,E2 16417.992} C_VEL
LIN {X 0,Y 560.198,Z 599.41,A -85,B 0,C 180,E1 16414.622,E2 16414.622} C_VEL
LIN {X 0,Y 566.827,Z 457.468,A -85,B 0,C 180,E1 16412.43,E2 16412.43} C_VEL
LIN {X 0,Y 555.152,Z 440.103,A -85,B 0,C 180,E1 16410.226,E2 16410.226} C_VEL
LIN {X 0,Y 544.655,Z 425.47,A -85,B 0,C 180,E1 16408.062,E2 16408.062} C_VEL
LIN {X 0,Y 534.691,Z 412.183,A -85,B 0,C 180,E1 16405.801,E2 16405.801} C_VEL
LIN {X 0,Y 526.247,Z 401.675,A -85,B 0,C 180,E1 16403.695,E2 16403.695} C_VEL
LIN {X 0,Y 521.378,Z 395.757,A -85,B 0,C 180,E1 16402.376,E2 16402.376} C_VEL
LIN {X 0,Y 516.933,Z 390.374,A -85,B 0,C 180,E1 16401.087,E2 16401.087} C_VEL
LIN {X 0,Y 512.037,Z 384.68,A -85,B 0,C 180,E1 16399.567,E2 16399.567} C_VEL
LIN {X 0,Y 507.93,Z 379.829,A -85,B 0,C 180,E1 16398.181,E2 16398.181} C_VEL
LIN {X 0,Y 502.898,Z 374.436,A -85,B 0,C 180,E1 16396.34,E2 16396.34} C_VEL
LIN {X 0,Y 501.525,Z 372.798,A -85,B 0,C 180,E1 16395.792,E2 16395.792} C_VEL
LIN {X 0,Y 497.683,Z 369.048,A -85,B 0,C 180,E1 16394.188,E2 16394.188} C_VEL
LIN {X 0,Y 495.946,Z 366.723,A -85,B 0,C 180,E1 16393.347,E2 16393.347} C_VEL
LIN {X 0,Y 493.136,Z 362.334,A -85,B 0,C 180,E1 16390.633,E2 16390.633} C_VEL
LIN {X 0,Y 492.377,Z 361.023,A -85,B 0,C 180,E1 16389.704,E2 16389.704} C_VEL
LIN {X 0,Y 489.274,Z 355.763,A -85,B 0,C 180,E1 16384.454,E2 16384.454} C_VEL
LIN {X 0,Y 487.987,Z 354.484,A -85,B 0,C 180,E1 16380,E2 16380} C_VEL
LIN {X 0,Y 488.489,Z 355.039,A -85,B 0,C 180,E1 16375.656,E2 16375.656} C_VEL
LIN {X 0,Y 489.557,Z 356.365,A -85,B 0,C 180,E1 16373.033,E2 16373.033} C_VEL
LIN {X 0,Y 492.959,Z 361.947,A -85,B 0,C 180,E1 16367.822,E2 16367.822} C_VEL
LIN {X 0,Y 495.433,Z 366.277,A -85,B 0,C 180,E1 16365.148,E2 16365.148} C_VEL
LIN {X 0,Y 496.289,Z 367.779,A -85,B 0,C 180,E1 16364.337,E2 16364.337} C_VEL
LIN {X 0,Y 498.82,Z 371.853,A -85,B 0,C 180,E1 16362.261,E2 16362.261} C_VEL
LIN {X 0,Y 501.709,Z 376.993,A -85,B 0,C 180,E1 16360.074,E2 16360.074} C_VEL
LIN {X 0,Y 504.373,Z 381.665,A -85,B 0,C 180,E1 16358.423,E2 16358.423} C_VEL
LIN {X 0,Y 510.826,Z 389.731,A -85,B 0,C 180,E1 16356.159,E2 16356.159} C_VEL
LIN {X 0,Y 518.651,Z 399.813,A -85,B 0,C 180,E1 16353.74,E2 16353.74} C_VEL
LIN {X 0,Y 525.695,Z 409.095,A -85,B 0,C 180,E1 16351.793,E2 16351.793} C_VEL
LIN {X 0,Y 534.356,Z 420.926,A -85,B 0,C 180,E1 16349.622,E2 16349.622} C_VEL
LIN {X 0,Y 544.719,Z 435.837,A -85,B 0,C 180,E1 16347.276,E2 16347.276} C_VEL
LIN {X 0,Y 556.472,Z 453.826,A -85,B 0,C 180,E1 16344.87,E2 16344.87} C_VEL
LIN {X 0,Y 563.175,Z 464.881,A -85,B 0,C 180,E1 16343.59,E2 16343.59} C_VEL
LIN {X 0,Y 553.274,Z 695.242,A -85,B 0,C 180,E1 16340.211,E2 16340.211} C_VEL
LIN {X 0,Y 547.682,Z 831.008,A -85,B 0,C 180,E1 16338.226,E2 16338.226} C_VEL
LIN {X 0,Y 545.565,Z 857.584,A -85,B 0,C 180,E1 16337.711,E2 16337.711} C_VEL
LIN {X 0,Y 542.865,Z 881.14,A -85,B 0,C 180,E1 16337.085,E2 16337.085} C_VEL
LIN {X 0,Y 540.286,Z 899.983,A -85,B 0,C 180,E1 16336.468,E2 16336.468} C_VEL
LIN {X 0,Y 537.161,Z 919.678,A -85,B 0,C 180,E1 16335.702,E2 16335.702} C_VEL
LIN {X 0,Y 532.842,Z 943.939,A -85,B 0,C 180,E1 16334.573,E2 16334.573} C_VEL
LIN {X 0,Y 528.258,Z 966.043,A -85,B 0,C 180,E1 16333.325,E2 16333.325} C_VEL
LIN {X 0,Y 523.94,Z 985.296,A -85,B 0,C 180,E1 16332.066,E2 16332.066} C_VEL
LIN {X 0,Y 518.953,Z 1006.237,A -85,B 0,C 180,E1 16330.489,E2 16330.489} C_VEL
LIN {X 0,Y 516.537,Z 1015.623,A -85,B 0,C 180,E1 16329.69,E2 16329.69} C_VEL
LIN {X 0,Y 514.179,Z 1021.865,A -85,B 0,C 180,E1 16329.225,E2 16329.225} C_VEL
LIN {X 0,Y 505.319,Z 1037.372,A -85,B 0,C 180,E1 16328.183,E2 16328.183} C_VEL
LIN {X 0,Y 502.947,Z 1042.969,A -85,B 0,C 180,E1 16327.654,E2 16327.654} C_VEL
LIN {X 0,Y 498.35,Z 1059.222,A -85,B 0,C 180,E1 16325.793,E2 16325.793} C_VEL
LIN {X 0,Y 492.943,Z 1078.092,A -85,B 0,C 180,E1 16323.31,E2 16323.31} C_VEL
LIN {X 0,Y 488.673,Z 1092.974,A -85,B 0,C 180,E1 16321.039,E2 16321.039} C_VEL
LIN {X 0,Y 485.141,Z 1105.738,A -85,B 0,C 180,E1 16318.834,E2 16318.834} C_VEL
LIN {X 0,Y 481.354,Z 1120.099,A -85,B 0,C 180,E1 16315.995,E2 16315.995} C_VEL
LIN {X 0,Y 478.455,Z 1131.851,A -85,B 0,C 180,E1 16313.265,E2 16313.265} C_VEL
LIN {X 0,Y 476.386,Z 1141.185,A -85,B 0,C 180,E1 16310.776,E2 16310.776} C_VEL
LIN {X 0,Y 474.503,Z 1151.165,A -85,B 0,C 180,E1 16307.664,E2 16307.664} C_VEL
LIN {X 0,Y 473.317,Z 1158.635,A -85,B 0,C 180,E1 16304.81,E2 16304.81} C_VEL
LIN {X 0,Y 472.632,Z 1164.293,A -85,B 0,C 180,E1 16302.204,E2 16302.204} C_VEL
LIN {X 0,Y 472.212,Z 1169.267,A -85,B 0,C 180,E1 16299.34,E2 16299.34} C_VEL
LIN {X 0,Y 471.983,Z 1173.255,A -85,B 0,C 180,E1 16296.081,E2 16296.081} C_VEL
LIN {X 0,Y 471.931,Z 1175.206,A -85,B 0,C 180,E1 16293.523,E2 16293.523} C_VEL
LIN {X 0,Y 471.929,Z 1176.111,A -85,B 0,C 180,E1 16291.093,E2 16291.093} C_VEL
LIN {X 0,Y 471.93,Z 1176.062,A -85,B 0,C 180,E1 16288.543,E2 16288.543} C_VEL
LIN {X 0,Y 471.94,Z 1174.799,A -85,B 0,C 180,E1 16285.626,E2 16285.626} C_VEL
LIN {X 0,Y 472.05,Z 1171.911,A -85,B 0,C 180,E1 16282.576,E2 16282.576} C_VEL
LIN {X 0,Y 472.267,Z 1168.192,A -85,B 0,C 180,E1 16279.903,E2 16279.903} C_VEL
LIN {X 0,Y 472.725,Z 1163.476,A -85,B 0,C 180,E1 16277.293,E2 16277.293} C_VEL
LIN {X 0,Y 473.657,Z 1156.504,A -85,B 0,C 180,E1 16274.198,E2 16274.198} C_VEL
LIN {X 0,Y 475.045,Z 1148.017,A -85,B 0,C 180,E1 16271.214,E2 16271.214} C_VEL
LIN {X 0,Y 476.772,Z 1139.35,A -85,B 0,C 180,E1 16268.617,E2 16268.617} C_VEL
LIN {X 0,Y 479.468,Z 1127.687,A -85,B 0,C 180,E1 16265.613,E2 16265.613} C_VEL
LIN {X 0,Y 482.623,Z 1115.107,A -85,B 0,C 180,E1 16262.885,E2 16262.885} C_VEL
LIN {X 0,Y 485.941,Z 1102.812,A -85,B 0,C 180,E1 16260.543,E2 16260.543} C_VEL
LIN {X 0,Y 490.309,Z 1087.48,A -85,B 0,C 180,E1 16257.981,E2 16257.981} C_VEL
LIN {X 0,Y 495.093,Z 1070.57,A -85,B 0,C 180,E1 16255.565,E2 16255.565} C_VEL
LIN {X 0,Y 499.428,Z 1055.437,A -85,B 0,C 180,E1 16253.658,E2 16253.658} C_VEL
LIN {X 0,Y 504.867,Z 1036.379,A -85,B 0,C 180,E1 16251.548,E2 16251.548} C_VEL
LIN {X 0,Y 510.213,Z 1016.521,A -85,B 0,C 180,E1 16249.672,E2 16249.672} C_VEL
LIN {X 0,Y 514.743,Z 999.021,A -85,B 0,C 180,E1 16248.221,E2 16248.221} C_VEL
LIN {X 0,Y 519.864,Z 978.189,A -85,B 0,C 180,E1 16246.712,E2 16246.712} C_VEL
LIN {X 0,Y 524.846,Z 955.714,A -85,B 0,C 180,E1 16245.334,E2 16245.334} C_VEL
LIN {X 0,Y 528.8,Z 936.015,A -85,B 0,C 180,E1 16244.301,E2 16244.301} C_VEL
LIN {X 0,Y 532.463,Z 915.681,A -85,B 0,C 180,E1 16243.388,E2 16243.388} C_VEL
LIN {X 0,Y 536.469,Z 890.137,A -85,B 0,C 180,E1 16242.443,E2 16242.443} C_VEL
LIN {X 0,Y 539.468,Z 866,A -85,B 0,C 180,E1 16241.749,E2 16241.749} C_VEL
LIN {X 0,Y 541.655,Z 844.082,A -85,B 0,C 180,E1 16241.262,E2 16241.262} C_VEL
LIN {X 0,Y 543.458,Z 815.866,A -85,B 0,C 180,E1 16240.789,E2 16240.789} C_VEL
LIN {X 0,Y 553.323,Z 582.92,A -85,B 0,C 180,E1 16237.381,E2 16237.381} C_VEL
LIN {X 0,Y 558.496,Z 468.675,A -85,B 0,C 180,E1 16235.676,E2 16235.676} C_VEL
LIN {X 0,Y 548.28,Z 452.344,A -85,B 0,C 180,E1 16233.638,E2 16233.638} C_VEL
LIN {X 0,Y 538.821,Z 438.043,A -85,B 0,C 180,E1 16231.586,E2 16231.586} C_VEL
LIN {X 0,Y 529.33,Z 424.433,A -85,B 0,C 180,E1 16229.322,E2 16229.322} C_VEL
LIN {X 0,Y 521.541,Z 413.677,A -85,B 0,C 180,E1 16227.272,E2 16227.272} C_VEL
LIN {X 0,Y 514.147,Z 403.92,A -85,B 0,C 180,E1 16225.116,E2 16225.116} C_VEL
LIN {X 0,Y 507.085,Z 394.75,A -85,B 0,C 180,E1 16222.797,E2 16222.797} C_VEL
LIN {X 0,Y 502.196,Z 388.662,A -85,B 0,C 180,E1 16221.001,E2 16221.001} C_VEL
LIN {X 0,Y 498.126,Z 383.68,A -85,B 0,C 180,E1 16219.342,E2 16219.342} C_VEL
LIN {X 0,Y 494.638,Z 378.828,A -85,B 0,C 180,E1 16217.651,E2 16217.651} C_VEL
LIN {X 0,Y 491.944,Z 374.57,A -85,B 0,C 180,E1 16215.442,E2 16215.442} C_VEL
LIN {X 0,Y 491.138,Z 373.023,A -85,B 0,C 180,E1 16214.622,E2 16214.622} C_VEL
LIN {X 0,Y 488.634,Z 368.564,A -85,B 0,C 180,E1 16211.808,E2 16211.808} C_VEL
LIN {X 0,Y 485.125,Z 362.632,A -85,B 0,C 180,E1 16205.796,E2 16205.796} C_VEL
LIN {X 0,Y 484.003,Z 361.513,A -85,B 0,C 180,E1 16201.302,E2 16201.302} C_VEL
LIN {X 0,Y 484.562,Z 362.113,A -85,B 0,C 180,E1 16197.28,E2 16197.28} C_VEL
LIN {X 0,Y 485.43,Z 363.252,A -85,B 0,C 180,E1 16195.037,E2 16195.037} C_VEL
LIN {X 0,Y 488.873,Z 368.434,A -85,B 0,C 180,E1 16189.988,E2 16189.988} C_VEL
LIN {X 0,Y 492.627,Z 372.99,A -85,B 0,C 180,E1 16187.814,E2 16187.814} C_VEL
LIN {X 0,Y 495.315,Z 375.392,A -85,B 0,C 180,E1 16186.517,E2 16186.517} C_VEL
LIN {X 0,Y 498.646,Z 379.426,A -85,B 0,C 180,E1 16185.009,E2 16185.009} C_VEL
LIN {X 0,Y 500.895,Z 381.485,A -85,B 0,C 180,E1 16184.099,E2 16184.099} C_VEL
LIN {X 0,Y 504.795,Z 386.017,A -85,B 0,C 180,E1 16182.596,E2 16182.596} C_VEL
LIN {X 0,Y 506.452,Z 387.826,A -85,B 0,C 180,E1 16182.002,E2 16182.002} C_VEL
LIN {X 0,Y 510.867,Z 392.764,A -85,B 0,C 180,E1 16180.506,E2 16180.506} C_VEL
LIN {X 0,Y 515.375,Z 398.18,A -85,B 0,C 180,E1 16179.085,E2 16179.085} C_VEL
LIN {X 0,Y 521.686,Z 406.046,A -85,B 0,C 180,E1 16177.252,E2 16177.252} C_VEL
LIN {X 0,Y 529.449,Z 415.615,A -85,B 0,C 180,E1 16175.212,E2 16175.212} C_VEL
LIN {X 0,Y 540.249,Z 429.997,A -85,B 0,C 180,E1 16172.648,E2 16172.648} C_VEL
LIN {X 0,Y 550.735,Z 444.708,A -85,B 0,C 180,E1 16170.407,E2 16170.407} C_VEL
LIN {X 0,Y 561.709,Z 461.086,A -85,B 0,C 180,E1 16168.263,E2 16168.263} C_VEL
LIN {X 0,Y 562.197,Z 462.258,A -85,B 0,C 180,E1 16168.162,E2 16168.162} C_VEL
LIN {X 0,Y 551.86,Z 674.712,A -85,B 0,C 180,E1 16164.886,E2 16164.886} C_VEL
LIN {X 0,Y 544.653,Z 826.455,A -85,B 0,C 180,E1 16162.54,E2 16162.54} C_VEL
LIN {X 0,Y 542.331,Z 853.773,A -85,B 0,C 180,E1 16162.007,E2 16162.007} C_VEL
LIN {X 0,Y 539.152,Z 880.191,A -85,B 0,C 180,E1 16161.298,E2 16161.298} C_VEL
LIN {X 0,Y 536.12,Z 901.554,A -85,B 0,C 180,E1 16160.586,E2 16160.586} C_VEL
LIN {X 0,Y 532.756,Z 922.317,A -85,B 0,C 180,E1 16159.763,E2 16159.763} C_VEL
LIN {X 0,Y 528.354,Z 946.729,A -85,B 0,C 180,E1 16158.62,E2 16158.62} C_VEL
LIN {X 0,Y 523.184,Z 971.75,A -85,B 0,C 180,E1 16157.212,E2 16157.212} C_VEL
LIN {X 0,Y 518.719,Z 991.823,A -85,B 0,C 180,E1 16155.903,E2 16155.903} C_VEL
LIN {X 0,Y 514.083,Z 1011.539,A -85,B 0,C 180,E1 16154.442,E2 16154.442} C_VEL
LIN {X 0,Y 508.281,Z 1035.118,A -85,B 0,C 180,E1 16152.434,E2 16152.434} C_VEL
LIN {X 0,Y 503.257,Z 1054.567,A -85,B 0,C 180,E1 16150.518,E2 16150.518} C_VEL
LIN {X 0,Y 498.964,Z 1071.036,A -85,B 0,C 180,E1 16148.698,E2 16148.698} C_VEL
LIN {X 0,Y 494.578,Z 1087.931,A -85,B 0,C 180,E1 16146.612,E2 16146.612} C_VEL
LIN {X 0,Y 489.292,Z 1108.482,A -85,B 0,C 180,E1 16143.723,E2 16143.723} C_VEL
LIN {X 0,Y 485.859,Z 1122.261,A -85,B 0,C 180,E1 16141.515,E2 16141.515} C_VEL
LIN {X 0,Y 482.997,Z 1134.296,A -85,B 0,C 180,E1 16139.361,E2 16139.361} C_VEL
LIN {X 0,Y 480.448,Z 1145.546,A -85,B 0,C 180,E1 16137.114,E2 16137.114} C_VEL
LIN {X 0,Y 478.166,Z 1156.196,A -85,B 0,C 180,E1 16134.722,E2 16134.722} C_VEL
LIN {X 0,Y 475.922,Z 1167.978,A -85,B 0,C 180,E1 16131.701,E2 16131.701} C_VEL
LIN {X 0,Y 474.241,Z 1178.151,A -85,B 0,C 180,E1 16128.564,E2 16128.564} C_VEL
LIN {X 0,Y 473.256,Z 1185.379,A -85,B 0,C 180,E1 16125.941,E2 16125.941} C_VEL
LIN {X 0,Y 472.664,Z 1190.798,A -85,B 0,C 180,E1 16123.58,E2 16123.58} C_VEL
LIN {X 0,Y 472.238,Z 1195.678,A -85,B 0,C 180,E1 16120.985,E2 16120.985} C_VEL
LIN {X 0,Y 472.041,Z 1199.343,A -85,B 0,C 180,E1 16118.527,E2 16118.527} C_VEL
LIN {X 0,Y 471.946,Z 1202.072,A -85,B 0,C 180,E1 16116.081,E2 16116.081} C_VEL
LIN {X 0,Y 471.915,Z 1203.882,A -85,B 0,C 180,E1 16113.644,E2 16113.644} C_VEL
LIN {X 0,Y 471.913,Z 1204.78,A -85,B 0,C 180,E1 16111.214,E2 16111.214} C_VEL
LIN {X 0,Y 471.913,Z 1204.78,A -85,B 0,C 180,E1 16108.786,E2 16108.786} C_VEL
LIN {X 0,Y 471.915,Z 1203.871,A -85,B 0,C 180,E1 16106.337,E2 16106.337} C_VEL
LIN {X 0,Y 471.95,Z 1201.957,A -85,B 0,C 180,E1 16103.797,E2 16103.797} C_VEL
LIN {X 0,Y 472.056,Z 1199.022,A -85,B 0,C 180,E1 16101.228,E2 16101.228} C_VEL
LIN {X 0,Y 472.296,Z 1194.851,A -85,B 0,C 180,E1 16098.521,E2 16098.521} C_VEL
LIN {X 0,Y 472.951,Z 1188.162,A -85,B 0,C 180,E1 16095.178,E2 16095.178} C_VEL
LIN {X 0,Y 473.862,Z 1180.703,A -85,B 0,C 180,E1 16092.311,E2 16092.311} C_VEL
LIN {X 0,Y 475.108,Z 1172.621,A -85,B 0,C 180,E1 16089.681,E2 16089.681} C_VEL
LIN {X 0,Y 476.702,Z 1163.714,A -85,B 0,C 180,E1 16087.167,E2 16087.167} C_VEL
LIN {X 0,Y 478.848,Z 1153.002,A -85,B 0,C 180,E1 16084.523,E2 16084.523} C_VEL
LIN {X 0,Y 482.122,Z 1138.189,A -85,B 0,C 180,E1 16081.375,E2 16081.375} C_VEL
LIN {X 0,Y 485.345,Z 1124.483,A -85,B 0,C 180,E1 16078.862,E2 16078.862} C_VEL
LIN {X 0,Y 488.738,Z 1110.652,A -85,B 0,C 180,E1 16076.61,E2 16076.61} C_VEL
LIN {X 0,Y 492.926,Z 1094.281,A -85,B 0,C 180,E1 16074.233,E2 16074.233} C_VEL
LIN {X 0,Y 498.323,Z 1073.565,A -85,B 0,C 180,E1 16071.598,E2 16071.598} C_VEL
LIN {X 0,Y 502.674,Z 1056.844,A -85,B 0,C 180,E1 16069.724,E2 16069.724} C_VEL
LIN {X 0,Y 507.147,Z 1039.473,A -85,B 0,C 180,E1 16067.983,E2 16067.983} C_VEL
LIN {X 0,Y 512.175,Z 1019.54,A -85,B 0,C 180,E1 16066.208,E2 16066.208} C_VEL
LIN {X 0,Y 517.958,Z 995.164,A -85,B 0,C 180,E1 16064.333,E2 16064.333} C_VEL
LIN {X 0,Y 522.394,Z 975.379,A -85,B 0,C 180,E1 16063.016,E2 16063.016} C_VEL
LIN {X 0,Y 526.463,Z 956.006,A -85,B 0,C 180,E1 16061.883,E2 16061.883} C_VEL
LIN {X 0,Y 530.439,Z 935.277,A -85,B 0,C 180,E1 16060.823,E2 16060.823} C_VEL
LIN {X 0,Y 535.107,Z 908.182,A -85,B 0,C 180,E1 16059.66,E2 16059.66} C_VEL
LIN {X 0,Y 538.596,Z 884.215,A -85,B 0,C 180,E1 16058.829,E2 16058.829} C_VEL
LIN {X 0,Y 541.28,Z 862.542,A -85,B 0,C 180,E1 16058.216,E2 16058.216} C_VEL
LIN {X 0,Y 543.555,Z 840.108,A -85,B 0,C 180,E1 16057.711,E2 16057.711} C_VEL
LIN {X 0,Y 545.657,Z 808.11,A -85,B 0,C 180,E1 16057.164,E2 16057.164} C_VEL
LIN {X 0,Y 556.307,Z 581.365,A -85,B 0,C 180,E1 16053.681,E2 16053.681} C_VEL
LIN {X 0,Y 562.135,Z 461.812,A -85,B 0,C 180,E1 16051.83,E2 16051.83} C_VEL
LIN {X 0,Y 551.236,Z 445.509,A -85,B 0,C 180,E1 16049.713,E2 16049.713} C_VEL
LIN {X 0,Y 541.346,Z 431.596,A -85,B 0,C 180,E1 16047.62,E2 16047.62} C_VEL
LIN {X 0,Y 531.945,Z 418.94,A -85,B 0,C 180,E1 16045.437,E2 16045.437} C_VEL
LIN {X 0,Y 523.813,Z 408.704,A -85,B 0,C 180,E1 16043.364,E2 16043.364} C_VEL
LIN {X 0,Y 519.104,Z 402.908,A -85,B 0,C 180,E1 16042.062,E2 16042.062} C_VEL
LIN {X 0,Y 514.722,Z 397.56,A -85,B 0,C 180,E1 16040.764,E2 16040.764} C_VEL
LIN {X 0,Y 510.063,Z 392.059,A -85,B 0,C 180,E1 16039.288,E2 16039.288} C_VEL
LIN {X 0,Y 505.95,Z 387.068,A -85,B 0,C 180,E1 16037.868,E2 16037.868} C_VEL
LIN {X 0,Y 501.341,Z 382.175,A -85,B 0,C 180,E1 16036.154,E2 16036.154} C_VEL
LIN {X 0,Y 499.85,Z 380.379,A -85,B 0,C 180,E1 16035.548,E2 16035.548} C_VEL
LIN {X 0,Y 496.075,Z 376.578,A -85,B 0,C 180,E1 16033.938,E2 16033.938} C_VEL
LIN {X 0,Y 494.555,Z 374.507,A -85,B 0,C 180,E1 16033.207,E2 16033.207} C_VEL
LIN {X 0,Y 489.83,Z 369.947,A -85,B 0,C 180,E1 16030.765,E2 16030.765} C_VEL
LIN {X 0,Y 488.421,Z 368.021,A -85,B 0,C 180,E1 16029.843,E2 16029.843} C_VEL
LIN {X 0,Y 485.092,Z 362.566,A -85,B 0,C 180,E1 16024.374,E2 16024.374} C_VEL
LIN {X 0,Y 483.841,Z 361.321,A -85,B 0,C 180,E1 16019.882,E2 16019.882} C_VEL
LIN {X 0,Y 484.391,Z 361.929,A -85,B 0,C 180,E1 16015.501,E2 16015.501} C_VEL
LIN {X 0,Y 485.348,Z 363.113,A -85,B 0,C 180,E1 16013.137,E2 16013.137} C_VEL
LIN {X 0,Y 488.631,Z 368.582,A -85,B 0,C 180,E1 16007.952,E2 16007.952} C_VEL
LIN {X 0,Y 491.045,Z 372.921,A -85,B 0,C 180,E1 16005.254,E2 16005.254} C_VEL
LIN {X 0,Y 491.884,Z 374.427,A -85,B 0,C 180,E1 16004.435,E2 16004.435} C_VEL
LIN {X 0,Y 494.866,Z 379.404,A -85,B 0,C 180,E1 16001.992,E2 16001.992} C_VEL
LIN {X 0,Y 498.428,Z 383.995,A -85,B 0,C 180,E1 16000.365,E2 16000.365} C_VEL
LIN {X 0,Y 504.07,Z 391.017,A -85,B 0,C 180,E1 15998.134,E2 15998.134} C_VEL
LIN {X 0,Y 509.063,Z 397.352,A -85,B 0,C 180,E1 15996.378,E2 15996.378} C_VEL
LIN {X 0,Y 516.455,Z 406.976,A -85,B 0,C 180,E1 15994.052,E2 15994.052} C_VEL
LIN {X 0,Y 523.401,Z 416.275,A -85,B 0,C 180,E1 15992.093,E2 15992.093} C_VEL
LIN {X 0,Y 531.858,Z 427.971,A -85,B 0,C 180,E1 15989.932,E2 15989.932} C_VEL
LIN {X 0,Y 541.993,Z 442.774,A -85,B 0,C 180,E1 15987.593,E2 15987.593} C_VEL
LIN {X 0,Y 553.27,Z 460.239,A -85,B 0,C 180,E1 15985.237,E2 15985.237} C_VEL
LIN {X 0,Y 558.501,Z 469.064,A -85,B 0,C 180,E1 15984.209,E2 15984.209} C_VEL
LIN {X 0,Y 548.252,Z 698.755,A -85,B 0,C 180,E1 15980.823,E2 15980.823} C_VEL
LIN {X 0,Y 542.583,Z 831.075,A -85,B 0,C 180,E1 15978.877,E2 15978.877} C_VEL
LIN {X 0,Y 540.384,Z 857.767,A -85,B 0,C 180,E1 15978.357,E2 15978.357} C_VEL
LIN {X 0,Y 537.637,Z 881.046,A -85,B 0,C 180,E1 15977.738,E2 15977.738} C_VEL
LIN {X 0,Y 534.834,Z 900.827,A -85,B 0,C 180,E1 15977.087,E2 15977.087} C_VEL
LIN {X 0,Y 531.405,Z 921.69,A -85,B 0,C 180,E1 15976.264,E2 15976.264} C_VEL
LIN {X 0,Y 526.543,Z 947.412,A -85,B 0,C 180,E1 15975.028,E2 15975.028} C_VEL
LIN {X 0,Y 522.224,Z 967.476,A -85,B 0,C 180,E1 15973.877,E2 15973.877} C_VEL
LIN {X 0,Y 517.766,Z 986.639,A -85,B 0,C 180,E1 15972.607,E2 15972.607} C_VEL
LIN {X 0,Y 512.274,Z 1008.764,A -85,B 0,C 180,E1 15970.908,E2 15970.908} C_VEL
LIN {X 0,Y 507.232,Z 1027.533,A -85,B 0,C 180,E1 15969.221,E2 15969.221} C_VEL
LIN {X 0,Y 502.947,Z 1042.969,A -85,B 0,C 180,E1 15967.654,E2 15967.654} C_VEL
LIN {X 0,Y 500.574,Z 1048.724,A -85,B 0,C 180,E1 15967.108,E2 15967.108} C_VEL
LIN {X 0,Y 491.109,Z 1063.836,A -85,B 0,C 180,E1 15965.778,E2 15965.778} C_VEL
LIN {X 0,Y 489.126,Z 1068.218,A -85,B 0,C 180,E1 15965.252,E2 15965.252} C_VEL
LIN {X 0,Y 484.642,Z 1083.17,A -85,B 0,C 180,E1 15963.143,E2 15963.143} C_VEL
LIN {X 0,Y 479.937,Z 1099.283,A -85,B 0,C 180,E1 15960.553,E2 15960.553} C_VEL
LIN {X 0,Y 475.903,Z 1113.169,A -85,B 0,C 180,E1 15957.939,E2 15957.939} C_VEL
LIN {X 0,Y 472.889,Z 1124.302,A -85,B 0,C 180,E1 15955.553,E2 15955.553} C_VEL
LIN {X 0,Y 469.958,Z 1136.145,A -85,B 0,C 180,E1 15952.65,E2 15952.65} C_VEL
LIN {X 0,Y 467.647,Z 1146.483,A -85,B 0,C 180,E1 15949.614,E2 15949.614} C_VEL
LIN {X 0,Y 466.189,Z 1154.222,A -85,B 0,C 180,E1 15946.943,E2 15946.943} C_VEL
LIN {X 0,Y 465.121,Z 1161.258,A -85,B 0,C 180,E1 15944.059,E2 15944.059} C_VEL
LIN {X 0,Y 464.4,Z 1167.499,A -85,B 0,C 180,E1 15940.796,E2 15940.796} C_VEL
LIN {X 0,Y 464.121,Z 1171.304,A -85,B 0,C 180,E1 15938.175,E2 15938.175} C_VEL
LIN {X 0,Y 463.971,Z 1174.059,A -85,B 0,C 180,E1 15935.565,E2 15935.565} C_VEL
LIN {X 0,Y 463.936,Z 1175.849,A -85,B 0,C 180,E1 15932.842,E2 15932.842} C_VEL
LIN {X 0,Y 463.922,Z 1176.507,A -85,B 0,C 180,E1 15929.63,E2 15929.63} C_VEL
LIN {X 0,Y 463.933,Z 1175.702,A -85,B 0,C 180,E1 15926.788,E2 15926.788} C_VEL
LIN {X 0,Y 463.976,Z 1173.922,A -85,B 0,C 180,E1 15924.187,E2 15924.187} C_VEL
LIN {X 0,Y 464.134,Z 1171.111,A -85,B 0,C 180,E1 15921.577,E2 15921.577} C_VEL
LIN {X 0,Y 464.526,Z 1166.242,A -85,B 0,C 180,E1 15918.347,E2 15918.347} C_VEL
LIN {X 0,Y 465.281,Z 1160.013,A -85,B 0,C 180,E1 15915.311,E2 15915.311} C_VEL
LIN {X 0,Y 466.335,Z 1153.405,A -85,B 0,C 180,E1 15912.661,E2 15912.661} C_VEL
LIN {X 0,Y 468.189,Z 1144.017,A -85,B 0,C 180,E1 15909.498,E2 15909.498} C_VEL
LIN {X 0,Y 470.682,Z 1133.008,A -85,B 0,C 180,E1 15906.461,E2 15906.461} C_VEL
LIN {X 0,Y 473.371,Z 1122.465,A -85,B 0,C 180,E1 15903.938,E2 15903.938} C_VEL
LIN {X 0,Y 477.254,Z 1108.581,A -85,B 0,C 180,E1 15901.056,E2 15901.056} C_VEL
LIN {X 0,Y 481.266,Z 1094.579,A -85,B 0,C 180,E1 15898.569,E2 15898.569} C_VEL
LIN {X 0,Y 485.228,Z 1081.257,A -85,B 0,C 180,E1 15896.479,E2 15896.479} C_VEL
LIN {X 0,Y 490.568,Z 1063.708,A -85,B 0,C 180,E1 15894.056,E2 15894.056} C_VEL
LIN {X 0,Y 495.904,Z 1045.475,A -85,B 0,C 180,E1 15891.904,E2 15891.904} C_VEL
LIN {X 0,Y 500.629,Z 1029.108,A -85,B 0,C 180,E1 15890.207,E2 15890.207} C_VEL
LIN {X 0,Y 505.597,Z 1011.304,A -85,B 0,C 180,E1 15888.578,E2 15888.578} C_VEL
LIN {X 0,Y 511.556,Z 988.468,A -85,B 0,C 180,E1 15886.779,E2 15886.779} C_VEL
LIN {X 0,Y 516.318,Z 968.71,A -85,B 0,C 180,E1 15885.452,E2 15885.452} C_VEL
LIN {X 0,Y 520.623,Z 949.45,A -85,B 0,C 180,E1 15884.332,E2 15884.332} C_VEL
LIN {X 0,Y 525.479,Z 925.291,A -85,B 0,C 180,E1 15883.137,E2 15883.137} C_VEL
LIN {X 0,Y 529.433,Z 902.033,A -85,B 0,C 180,E1 15882.201,E2 15882.201} C_VEL
LIN {X 0,Y 532.3,Z 882.601,A -85,B 0,C 180,E1 15881.553,E2 15881.553} C_VEL
LIN {X 0,Y 534.871,Z 861.696,A -85,B 0,C 180,E1 15880.982,E2 15880.982} C_VEL
LIN {X 0,Y 537.421,Z 834.275,A -85,B 0,C 180,E1 15880.417,E2 15880.417} C_VEL
LIN {X 0,Y 539.968,Z 780.442,A -85,B 0,C 180,E1 15879.605,E2 15879.605} C_VEL
LIN {X 0,Y 549.984,Z 555.661,A -85,B 0,C 180,E1 15876.29,E2 15876.29} C_VEL
LIN {X 0,Y 553.851,Z 472.715,A -85,B 0,C 180,E1 15875.037,E2 15875.037} C_VEL
LIN {X 0,Y 542.734,Z 454.891,A -85,B 0,C 180,E1 15872.733,E2 15872.733} C_VEL
LIN {X 0,Y 532.616,Z 439.711,A -85,B 0,C 180,E1 15870.425,E2 15870.425} C_VEL
LIN {X 0,Y 523.597,Z 426.754,A -85,B 0,C 180,E1 15868.144,E2 15868.144} C_VEL
LIN {X 0,Y 516.406,Z 416.996,A -85,B 0,C 180,E1 15866.136,E2 15866.136} C_VEL
LIN {X 0,Y 511.563,Z 410.541,A -85,B 0,C 180,E1 15864.658,E2 15864.658} C_VEL
LIN {X 0,Y 505.206,Z 402.143,A -85,B 0,C 180,E1 15862.518,E2 15862.518} C_VEL
LIN {X 0,Y 500.396,Z 396.052,A -85,B 0,C 180,E1 15860.713,E2 15860.713} C_VEL
LIN {X 0,Y 496.393,Z 391.114,A -85,B 0,C 180,E1 15859.046,E2 15859.046} C_VEL
LIN {X 0,Y 492.341,Z 385.829,A -85,B 0,C 180,E1 15857.126,E2 15857.126} C_VEL
LIN {X 0,Y 488.729,Z 381.57,A -85,B 0,C 180,E1 15855.181,E2 15855.181} C_VEL
LIN {X 0,Y 487.392,Z 379.945,A -85,B 0,C 180,E1 15854.373,E2 15854.373} C_VEL
LIN {X 0,Y 484.505,Z 375.832,A -85,B 0,C 180,E1 15852.031,E2 15852.031} C_VEL
LIN {X 0,Y 483.702,Z 374.391,A -85,B 0,C 180,E1 15850.963,E2 15850.963} C_VEL
LIN {X 0,Y 480.936,Z 369.435,A -85,B 0,C 180,E1 15845.727,E2 15845.727} C_VEL
LIN {X 0,Y 479.856,Z 368.352,A -85,B 0,C 180,E1 15841.194,E2 15841.194} C_VEL
LIN {X 0,Y 480.468,Z 369.007,A -85,B 0,C 180,E1 15837.137,E2 15837.137} C_VEL
LIN {X 0,Y 481.334,Z 370.093,A -85,B 0,C 180,E1 15835.114,E2 15835.114} C_VEL
LIN {X 0,Y 487.812,Z 376.66,A -85,B 0,C 180,E1 15829.966,E2 15829.966} C_VEL
LIN {X 0,Y 491.649,Z 381.069,A -85,B 0,C 180,E1 15827.789,E2 15827.789} C_VEL
LIN {X 0,Y 493.847,Z 383.105,A -85,B 0,C 180,E1 15826.714,E2 15826.714} C_VEL
LIN {X 0,Y 497.27,Z 387.221,A -85,B 0,C 180,E1 15825.145,E2 15825.145} C_VEL
LIN {X 0,Y 499.287,Z 389.136,A -85,B 0,C 180,E1 15824.314,E2 15824.314} C_VEL
LIN {X 0,Y 503.216,Z 393.694,A -85,B 0,C 180,E1 15822.779,E2 15822.779} C_VEL
LIN {X 0,Y 504.845,Z 395.599,A -85,B 0,C 180,E1 15822.182,E2 15822.182} C_VEL
LIN {X 0,Y 509.844,Z 401.477,A -85,B 0,C 180,E1 15820.465,E2 15820.465} C_VEL
LIN {X 0,Y 514.701,Z 407.342,A -85,B 0,C 180,E1 15818.937,E2 15818.937} C_VEL
LIN {X 0,Y 519.579,Z 413.414,A -85,B 0,C 180,E1 15817.513,E2 15817.513} C_VEL
LIN {X 0,Y 527.06,Z 422.75,A -85,B 0,C 180,E1 15815.511,E2 15815.511} C_VEL
LIN {X 0,Y 537.527,Z 436.856,A -85,B 0,C 180,E1 15812.977,E2 15812.977} C_VEL
LIN {X 0,Y 547.889,Z 451.585,A -85,B 0,C 180,E1 15810.719,E2 15810.719} C_VEL
LIN {X 0,Y 557.543,Z 466.21,A -85,B 0,C 180,E1 15808.786,E2 15808.786} C_VEL
LIN {X 0,Y 546.845,Z 678.75,A -85,B 0,C 180,E1 15805.494,E2 15805.494} C_VEL
LIN {X 0,Y 539.573,Z 826.561,A -85,B 0,C 180,E1 15803.196,E2 15803.196} C_VEL
LIN {X 0,Y 537.17,Z 853.973,A -85,B 0,C 180,E1 15802.659,E2 15802.659} C_VEL
LIN {X 0,Y 533.912,Z 880.259,A -85,B 0,C 180,E1 15801.951,E2 15801.951} C_VEL
LIN {X 0,Y 530.818,Z 901.414,A -85,B 0,C 180,E1 15801.245,E2 15801.245} C_VEL
LIN {X 0,Y 527.246,Z 922.754,A -85,B 0,C 180,E1 15800.396,E2 15800.396} C_VEL
LIN {X 0,Y 522.478,Z 948.25,A -85,B 0,C 180,E1 15799.189,E2 15799.189} C_VEL
LIN {X 0,Y 517.352,Z 972.065,A -85,B 0,C 180,E1 15797.832,E2 15797.832} C_VEL
LIN {X 0,Y 512.83,Z 991.704,A -85,B 0,C 180,E1 15796.543,E2 15796.543} C_VEL
LIN {X 0,Y 508.129,Z 1010.998,A -85,B 0,C 180,E1 15795.104,E2 15795.104} C_VEL
LIN {X 0,Y 502.258,Z 1033.996,A -85,B 0,C 180,E1 15793.143,E2 15793.143} C_VEL
LIN {X 0,Y 496.847,Z 1054.076,A -85,B 0,C 180,E1 15791.152,E2 15791.152} C_VEL
LIN {X 0,Y 492.334,Z 1070.636,A -85,B 0,C 180,E1 15789.305,E2 15789.305} C_VEL
LIN {X 0,Y 487.898,Z 1086.94,A -85,B 0,C 180,E1 15787.271,E2 15787.271} C_VEL
LIN {X 0,Y 482.772,Z 1106.036,A -85,B 0,C 180,E1 15784.575,E2 15784.575} C_VEL
LIN {X 0,Y 478.436,Z 1122.387,A -85,B 0,C 180,E1 15781.92,E2 15781.92} C_VEL
LIN {X 0,Y 475.402,Z 1134.587,A -85,B 0,C 180,E1 15779.698,E2 15779.698} C_VEL
LIN {X 0,Y 472.653,Z 1146.271,A -85,B 0,C 180,E1 15777.314,E2 15777.314} C_VEL
LIN {X 0,Y 469.787,Z 1159.484,A -85,B 0,C 180,E1 15774.253,E2 15774.253} C_VEL
LIN {X 0,Y 467.612,Z 1170.571,A -85,B 0,C 180,E1 15771.184,E2 15771.184} C_VEL
LIN {X 0,Y 466.243,Z 1178.701,A -85,B 0,C 180,E1 15768.576,E2 15768.576} C_VEL
LIN {X 0,Y 465.298,Z 1185.369,A -85,B 0,C 180,E1 15766.093,E2 15766.093} C_VEL
LIN {X 0,Y 464.662,Z 1191.126,A -85,B 0,C 180,E1 15763.565,E2 15763.565} C_VEL
LIN {X 0,Y 464.236,Z 1196.063,A -85,B 0,C 180,E1 15760.925,E2 15760.925} C_VEL
LIN {X 0,Y 464.036,Z 1199.66,A -85,B 0,C 180,E1 15758.425,E2 15758.425} C_VEL
LIN {X 0,Y 463.941,Z 1202.41,A -85,B 0,C 180,E1 15755.813,E2 15755.813} C_VEL
LIN {X 0,Y 463.915,Z 1204.356,A -85,B 0,C 180,E1 15752.841,E2 15752.841} C_VEL
LIN {X 0,Y 463.897,Z 1204.938,A -85,B 0,C 180,E1 15749.629,E2 15749.629} C_VEL
LIN {X 0,Y 463.915,Z 1204.151,A -85,B 0,C 180,E1 15746.787,E2 15746.787} C_VEL
LIN {X 0,Y 463.943,Z 1202.295,A -85,B 0,C 180,E1 15744.062,E2 15744.062} C_VEL
LIN {X 0,Y 464.04,Z 1199.572,A -85,B 0,C 180,E1 15741.507,E2 15741.507} C_VEL
LIN {X 0,Y 464.236,Z 1196.061,A -85,B 0,C 180,E1 15739.074,E2 15739.074} C_VEL
LIN {X 0,Y 464.662,Z 1191.128,A -85,B 0,C 180,E1 15736.435,E2 15736.435} C_VEL
LIN {X 0,Y 465.315,Z 1185.237,A -85,B 0,C 180,E1 15733.851,E2 15733.851} C_VEL
LIN {X 0,Y 466.333,Z 1178.176,A -85,B 0,C 180,E1 15731.239,E2 15731.239} C_VEL
LIN {X 0,Y 468.087,Z 1168.052,A -85,B 0,C 180,E1 15728.049,E2 15728.049} C_VEL
LIN {X 0,Y 470.427,Z 1156.289,A -85,B 0,C 180,E1 15724.978,E2 15724.978} C_VEL
LIN {X 0,Y 472.938,Z 1145.045,A -85,B 0,C 180,E1 15722.419,E2 15722.419} C_VEL
LIN {X 0,Y 475.82,Z 1132.887,A -85,B 0,C 180,E1 15719.972,E2 15719.972} C_VEL
LIN {X 0,Y 480.015,Z 1116.562,A -85,B 0,C 180,E1 15717.084,E2 15717.084} C_VEL
LIN {X 0,Y 484.558,Z 1099.148,A -85,B 0,C 180,E1 15714.415,E2 15714.415} C_VEL
LIN {X 0,Y 488.639,Z 1084.144,A -85,B 0,C 180,E1 15712.365,E2 15712.365} C_VEL
LIN {X 0,Y 493.376,Z 1066.874,A -85,B 0,C 180,E1 15710.253,E2 15710.253} C_VEL
LIN {X 0,Y 499.432,Z 1044.59,A -85,B 0,C 180,E1 15707.88,E2 15707.88} C_VEL
LIN {X 0,Y 504.331,Z 1025.899,A -85,B 0,C 180,E1 15706.144,E2 15706.144} C_VEL
LIN {X 0,Y 508.885,Z 1007.943,A -85,B 0,C 180,E1 15704.661,E2 15704.661} C_VEL
LIN {X 0,Y 513.683,Z 988.144,A -85,B 0,C 180,E1 15703.214,E2 15703.214} C_VEL
LIN {X 0,Y 519.503,Z 962.341,A -85,B 0,C 180,E1 15701.591,E2 15701.591} C_VEL
LIN {X 0,Y 523.979,Z 940.186,A -85,B 0,C 180,E1 15700.413,E2 15700.413} C_VEL
LIN {X 0,Y 527.793,Z 919.469,A -85,B 0,C 180,E1 15699.467,E2 15699.467} C_VEL
LIN {X 0,Y 531.519,Z 896.798,A -85,B 0,C 180,E1 15698.59,E2 15698.59} C_VEL
LIN {X 0,Y 535.472,Z 868.043,A -85,B 0,C 180,E1 15697.702,E2 15697.702} C_VEL
LIN {X 0,Y 537.974,Z 845.146,A -85,B 0,C 180,E1 15697.159,E2 15697.159} C_VEL
LIN {X 0,Y 539.789,Z 822.652,A -85,B 0,C 180,E1 15696.741,E2 15696.741} C_VEL
LIN {X 0,Y 550.349,Z 607.088,A -85,B 0,C 180,E1 15693.401,E2 15693.401} C_VEL
LIN {X 0,Y 557.389,Z 465.97,A -85,B 0,C 180,E1 15691.197,E2 15691.197} C_VEL
LIN {X 0,Y 546.415,Z 449.493,A -85,B 0,C 180,E1 15688.992,E2 15688.992} C_VEL
LIN {X 0,Y 535.872,Z 434.557,A -85,B 0,C 180,E1 15686.664,E2 15686.664} C_VEL
LIN {X 0,Y 525.879,Z 421.337,A -85,B 0,C 180,E1 15684.219,E2 15684.219} C_VEL
LIN {X 0,Y 517.574,Z 410.83,A -85,B 0,C 180,E1 15681.951,E2 15681.951} C_VEL
LIN {X 0,Y 512.528,Z 404.738,A -85,B 0,C 180,E1 15680.439,E2 15680.439} C_VEL
LIN {X 0,Y 508.102,Z 399.434,A -85,B 0,C 180,E1 15679.007,E2 15679.007} C_VEL
LIN {X 0,Y 503.216,Z 393.695,A -85,B 0,C 180,E1 15677.281,E2 15677.281} C_VEL
LIN {X 0,Y 499.197,Z 389.025,A -85,B 0,C 180,E1 15675.718,E2 15675.718} C_VEL
LIN {X 0,Y 494.245,Z 383.764,A -85,B 0,C 180,E1 15673.573,E2 15673.573} C_VEL
LIN {X 0,Y 492.855,Z 382.027,A -85,B 0,C 180,E1 15672.895,E2 15672.895} C_VEL
LIN {X 0,Y 488.355,Z 377.489,A -85,B 0,C 180,E1 15670.499,E2 15670.499} C_VEL
LIN {X 0,Y 487.065,Z 375.821,A -85,B 0,C 180,E1 15669.691,E2 15669.691} C_VEL
LIN {X 0,Y 481.699,Z 370.637,A -85,B 0,C 180,E1 15665.599,E2 15665.599} C_VEL
LIN {X 0,Y 480.739,Z 369.21,A -85,B 0,C 180,E1 15663.936,E2 15663.936} C_VEL
LIN {X 0,Y 479.68,Z 368.143,A -85,B 0,C 180,E1 15659.522,E2 15659.522} C_VEL
LIN {X 0,Y 480.422,Z 368.949,A -85,B 0,C 180,E1 15654.985,E2 15654.985} C_VEL
LIN {X 0,Y 481.183,Z 370.034,A -85,B 0,C 180,E1 15653.078,E2 15653.078} C_VEL
LIN {X 0,Y 484.367,Z 375.431,A -85,B 0,C 180,E1 15647.966,E2 15647.966} C_VEL
LIN {X 0,Y 486.312,Z 378.872,A -85,B 0,C 180,E1 15646.08,E2 15646.08} C_VEL
LIN {X 0,Y 488.59,Z 381.399,A -85,B 0,C 180,E1 15644.693,E2 15644.693} C_VEL
LIN {X 0,Y 492.215,Z 385.749,A -85,B 0,C 180,E1 15642.747,E2 15642.747} C_VEL
LIN {X 0,Y 493.946,Z 388.069,A -85,B 0,C 180,E1 15641.897,E2 15641.897} C_VEL
LIN {X 0,Y 498.124,Z 393.266,A -85,B 0,C 180,E1 15640.047,E2 15640.047} C_VEL
LIN {X 0,Y 502.306,Z 398.508,A -85,B 0,C 180,E1 15638.391,E2 15638.391} C_VEL
LIN {X 0,Y 507.154,Z 404.738,A -85,B 0,C 180,E1 15636.654,E2 15636.654} C_VEL
LIN {X 0,Y 514.361,Z 414.264,A -85,B 0,C 180,E1 15634.341,E2 15634.341} C_VEL
LIN {X 0,Y 521.029,Z 423.311,A -85,B 0,C 180,E1 15632.421,E2 15632.421} C_VEL
LIN {X 0,Y 530.186,Z 436.152,A -85,B 0,C 180,E1 15630.046,E2 15630.046} C_VEL
LIN {X 0,Y 541.129,Z 452.519,A -85,B 0,C 180,E1 15627.504,E2 15627.504} C_VEL
LIN {X 0,Y 551.239,Z 468.561,A -85,B 0,C 180,E1 15625.375,E2 15625.375} C_VEL
LIN {X 0,Y 553.895,Z 473.13,A -85,B 0,C 180,E1 15624.84,E2 15624.84} C_VEL
LIN {X 0,Y 543.291,Z 702.278,A -85,B 0,C 180,E1 15621.447,E2 15621.447} C_VEL
LIN {X 0,Y 537.552,Z 831.171,A -85,B 0,C 180,E1 15619.54,E2 15619.54} C_VEL
LIN {X 0,Y 535.249,Z 858.134,A -85,B 0,C 180,E1 15619.01,E2 15619.01} C_VEL
